// TIA Portal V16 export
// export: Created 2021-11-12T13:32:15.9169285Z, ExportSetting WithDefaults, DisplayName Totally Integrated Automation Portal, DisplayVersion V16 Update 3, DisplayName TIA Portal Version Control Interface, DisplayVersion V16 Update 2, DisplayName TIA Portal Openness, DisplayVersion V16 Update 3, DisplayName SINAMICS Startdrive Advanced, DisplayVersion V16 Update 5, DisplayName SINAMICS Startdrive G130, G150, S120, S150, SINAMICS MV, S210, DisplayVersion V16 Update 5, DisplayName SINAMICS Startdrive G110M, G120, G120C, G120D, G120P, G115D, DisplayVersion V16 Update 5, DisplayName STEP 7 Professional, DisplayVersion V16 Update 3, DisplayName STEP 7 Safety, DisplayVersion V16, DisplayName WinCC UA Professional, DisplayVersion V16 Update 3
FUNCTION_BLOCK "StationBSN2"   // FB15, LAD
{ S7_Optimized_Access := 'TRUE' }
VERSION : 0.1
// stored: AutoNumber true, IsIECCheckEnabled false, IsRetainMemResEnabled false, MemoryReserve 100, SetENOAutomatically false, UDAEnableTagReadback false
   VAR_INPUT
      IS_Inputs : "UDT_COMM_BSN2_CRS";
   END_VAR
   VAR_OUTPUT
      OS_Outputs : "UDT_COMM_CRS_BSN2";
      OS_Status : "UDT_BSN12_Status_specific";
   END_VAR
   VAR
      SF_Alarm1 : "STD_DI_Mon";
      SF_Alarm2 : "STD_DI_Mon";
      SF_Alarm3 : "STD_DI_Mon";
      SF_Alarm4 : "STD_DI_Mon";
      SF_Alarm5 : "STD_DI_Mon";
      SF_Alarm6 : "STD_DI_Mon";
      SF_Alarm7 : "STD_DI_Mon";
      SF_Alarm8 : "STD_DI_Mon";
      SS_Edge : Array[0..15] of Bool;   // Edge evalution
      SS_ParamTemp : Struct
         PartType : Int;   // Production type
         SPTactTime : Int := 0;   // setpoint tact time [s]
         SPStepLength : Int := 0;   // setpoint step length
         SPBurnerHigh : Int := 0;   // setpoint burner high [mm]
         SPTempSetpointZ1 : Int := 0;   // temperature setpoint in zone 1 [°C]
         SPTempSetpointZ2 : Int := 0;   // temperature setpoint in zone 2 [°C]
         SPTempSetpointZ3 : Int := 0;   // temperature setpoint in zone 3 [°C]
         SPTempSetpointZ4 : Int := 0;   // temperature setpoint in zone 4 [°C]
         SPTempSetpointZ5 : Int := 0;   // temperature setpoint in zone 5 [°C]
      END_STRUCT;
      SS_RobotZones : "STD_RobotZones";
      SDIPartID : DInt;
      SI_PartType : Int;
      SI_EjectPartPos { ExternalAccessible := 'False'; ExternalVisible := 'False'; ExternalWritable := 'False'} : Int;   // Position of ejected part
      SB1BlockMapMove : Bool;   // Block transfer datas in map when comm error
      SB1ReqBlockBeltMtion : Bool;   // Button request to block belt motion
      SB1ReqBlockBeltMtion_Aux : Bool;
      SB1ParamChanged : Bool;   // Production paramaters changed trigger
      SB1ReqOnePart { ExternalAccessible := 'False'; ExternalVisible := 'False'; ExternalWritable := 'False'} : Bool;   // Request to eject one part
      SB1ReqAllParts { ExternalAccessible := 'False'; ExternalVisible := 'False'; ExternalWritable := 'False'} : Bool;   // Request to eject all parts in row
      SB1PartEjected : Bool;   // Part ejected memory
      SB1RowEjected : Bool;   // Whole row ejected memory
      SF_TOF_ClearDelay { S7_SetPoint := 'True'} : TOF_TIME;
   END_VAR
   VAR_TEMP
      TS_ParamTemp : Struct
         PartType : Int;   // Production type
         SPTactTime : Int;   // setpoint tact time [s]
         SPStepLength : Int;   // setpoint step length
         SPBurnerHigh : Int;   // setpoint burner high [mm]
         SPTempSetpointZ1 : Int;   // temperature setpoint in zone 1 [°C]
         SPTempSetpointZ2 : Int;   // temperature setpoint in zone 2 [°C]
         SPTempSetpointZ3 : Int;   // temperature setpoint in zone 3 [°C]
         SPTempSetpointZ4 : Int;   // temperature setpoint in zone 4 [°C]
         SPTempSetpointZ5 : Int;   // temperature setpoint in zone 5 [°C]
      END_STRUCT;
      TS_CmdEject : Array[1..5] of Bool;
      TS_EjectSelPreset : Array[1..5] of Byte;
      TS_Part : "UDT_MatCard";
      TDITimeInFurnace_ms : DInt;
      TI_RowNr : Int;   // Transfer mat card according to row number
      TI_BufferFreePos : Int;   // Number of free position in buffer
      TB1PwrOk : Bool;
      TB1BeltMtionBlock : Bool;   // Belt motion blocking
      TB1ReqBlockBeltMtion : Bool;
      TB1SetParam : Bool;   // Set loaded parameters memory
      TB1FreePosBSN : Bool;   // Free position in furnace was found
   END_VAR
   VAR CONSTANT
      CI_FirstRowInsideOven : Int := 8;
      CI_LastRow : Int := 225;
   END_VAR
   // // IS_Inputs.Eject1Up : bsn2 - ejector 1 upper position
   // // IS_Inputs.Eject2Up : bsn2 - ejector 2 upper position
   // // IS_Inputs.Eject3Up : bsn2 - ejector 3 upper position
   // // IS_Inputs.Eject4Up : bsn2 - ejector 4 upper position
   // // IS_Inputs.Eject5Up : bsn2 - ejector 5 upper position
   // // TS_Part.TimeBSN4_s : Time in bsn2 (s)
   VAR_TEMP   // added for the SCL form of the ladder/FBD networks
      _w1 : Bool;
      _w2 : Bool;
      _w3 : Bool;
      _w4 : Bool;
      _w5 : Bool;
      _w6 : Bool;
      _w7 : Bool;
      _w8 : Bool;
      _w9 : Bool;
      _w10 : Bool;
      _w11 : Bool;
      _w12 : Bool;
      _w13 : Bool;
      _w14 : Bool;
      _w15 : Bool;
      _w16 : Bool;
      _w17 : Bool;
      _w18 : Bool;
      _w19 : Bool;
      _w20 : Bool;
      _w21 : Bool;
      _w22 : Bool;
      _w23 : Bool;
      _w24 : Bool;
      _w25 : Bool;
      _w26 : Bool;
   END_VAR
BEGIN

REGION Network 1: *************** Alarms ***************
END_REGION

REGION Network 2: Power OK
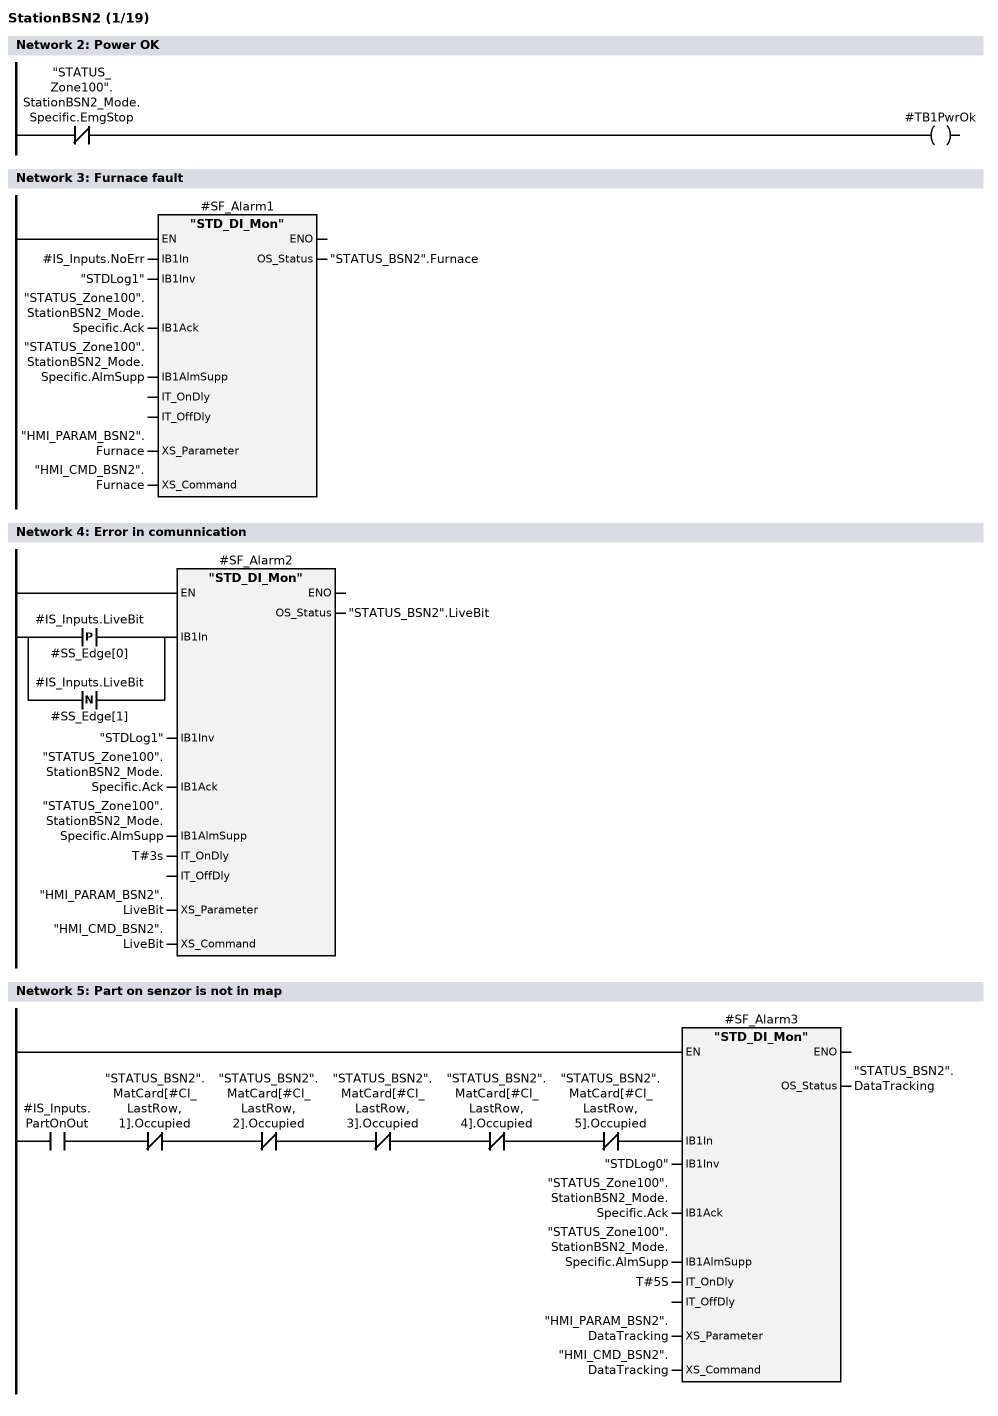
   RUNG wire#powerrail
      I_Contact( "STATUS_Zone100".StationBSN2_Mode.Specific.EmgStop )
      Coil( #TB1PwrOk )
   END_RUNG
   // the same network as SCL:
   #TB1PwrOk := NOT "STATUS_Zone100".StationBSN2_Mode.Specific.EmgStop;
END_REGION

REGION Network 3: Furnace fault
   RUNG wire#powerrail
      #SF_Alarm1(IB1In := #IS_Inputs.NoErr, IB1Inv := "STDLog1", IB1Ack := "STATUS_Zone100".StationBSN2_Mode.Specific.Ack, IB1AlmSupp := "STATUS_Zone100".StationBSN2_Mode.Specific.AlmSupp, IT_OnDly :=, IT_OffDly :=, XS_Parameter := "HMI_PARAM_BSN2".Furnace, XS_Command := "HMI_CMD_BSN2".Furnace, OS_Status => "STATUS_BSN2".Furnace)
   END_RUNG
   // the same network as SCL:
   #SF_Alarm1(IB1In := #IS_Inputs.NoErr,   // "STD_DI_Mon"
              IB1Inv := "STDLog1",
              IB1Ack := "STATUS_Zone100".StationBSN2_Mode.Specific.Ack,
              IB1AlmSupp := "STATUS_Zone100".StationBSN2_Mode.Specific.AlmSupp,
              XS_Parameter := "HMI_PARAM_BSN2".Furnace,
              XS_Command := "HMI_CMD_BSN2".Furnace,
              OS_Status => "STATUS_BSN2".Furnace);
END_REGION

REGION Network 4: Error in comunnication
   RUNG wire#powerrail
      #SF_Alarm2(IB1In := wire#w1, IB1Inv := "STDLog1", IB1Ack := "STATUS_Zone100".StationBSN2_Mode.Specific.Ack, IB1AlmSupp := "STATUS_Zone100".StationBSN2_Mode.Specific.AlmSupp, IT_OnDly := T#3s, IT_OffDly :=, XS_Parameter := "HMI_PARAM_BSN2".LiveBit, XS_Command := "HMI_CMD_BSN2".LiveBit, OS_Status => "STATUS_BSN2".LiveBit)
   END_RUNG
   RUNG wire#powerrail
      P_Contact(operand := #IS_Inputs.LiveBit, bit := #SS_Edge[0])
   END_RUNG wire#w1
   RUNG wire#powerrail
      N_Contact(operand := #IS_Inputs.LiveBit, bit := #SS_Edge[1])
   END_RUNG wire#w1
   // the same network as SCL:
   #_w1 := #IS_Inputs.LiveBit AND NOT #SS_Edge[0];   // rising edge of #IS_Inputs.LiveBit
   #SS_Edge[0] := #IS_Inputs.LiveBit;
   #_w2 := NOT #IS_Inputs.LiveBit AND #SS_Edge[1];   // falling edge of #IS_Inputs.LiveBit
   #SS_Edge[1] := #IS_Inputs.LiveBit;
   #SF_Alarm2(IB1In := #_w1 OR #_w2,   // "STD_DI_Mon"
              IB1Inv := "STDLog1",
              IB1Ack := "STATUS_Zone100".StationBSN2_Mode.Specific.Ack,
              IB1AlmSupp := "STATUS_Zone100".StationBSN2_Mode.Specific.AlmSupp,
              IT_OnDly := T#3s,
              XS_Parameter := "HMI_PARAM_BSN2".LiveBit,
              XS_Command := "HMI_CMD_BSN2".LiveBit,
              OS_Status => "STATUS_BSN2".LiveBit);
END_REGION

REGION Network 5: Part on senzor is not in map
   RUNG wire#powerrail
      #SF_Alarm3(IB1In := wire#w1, IB1Inv := "STDLog0", IB1Ack := "STATUS_Zone100".StationBSN2_Mode.Specific.Ack, IB1AlmSupp := "STATUS_Zone100".StationBSN2_Mode.Specific.AlmSupp, IT_OnDly := T#5S, IT_OffDly :=, XS_Parameter := "HMI_PARAM_BSN2".DataTracking, XS_Command := "HMI_CMD_BSN2".DataTracking, OS_Status => "STATUS_BSN2".DataTracking)
   END_RUNG
   RUNG wire#powerrail
      Contact( #IS_Inputs.PartOnOut )
      I_Contact( "STATUS_BSN2".MatCard[#CI_LastRow, 1].Occupied )
      I_Contact( "STATUS_BSN2".MatCard[#CI_LastRow, 2].Occupied )
      I_Contact( "STATUS_BSN2".MatCard[#CI_LastRow, 3].Occupied )
      I_Contact( "STATUS_BSN2".MatCard[#CI_LastRow, 4].Occupied )
      I_Contact( "STATUS_BSN2".MatCard[#CI_LastRow, 5].Occupied )
   END_RUNG wire#w1
   // the same network as SCL:
   #SF_Alarm3(IB1In := #IS_Inputs.PartOnOut AND NOT "STATUS_BSN2".MatCard[#CI_LastRow, 1].Occupied AND NOT "STATUS_BSN2".MatCard[#CI_LastRow, 2].Occupied AND NOT "STATUS_BSN2".MatCard[#CI_LastRow, 3].Occupied AND NOT "STATUS_BSN2".MatCard[#CI_LastRow, 4].Occupied AND NOT "STATUS_BSN2".MatCard[#CI_LastRow, 5].Occupied,   // "STD_DI_Mon"
              IB1Inv := "STDLog0",
              IB1Ack := "STATUS_Zone100".StationBSN2_Mode.Specific.Ack,
              IB1AlmSupp := "STATUS_Zone100".StationBSN2_Mode.Specific.AlmSupp,
              IT_OnDly := T#5S,
              XS_Parameter := "HMI_PARAM_BSN2".DataTracking,
              XS_Command := "HMI_CMD_BSN2".DataTracking,
              OS_Status => "STATUS_BSN2".DataTracking);
END_REGION

REGION Network 6: Part in map is not on senzor
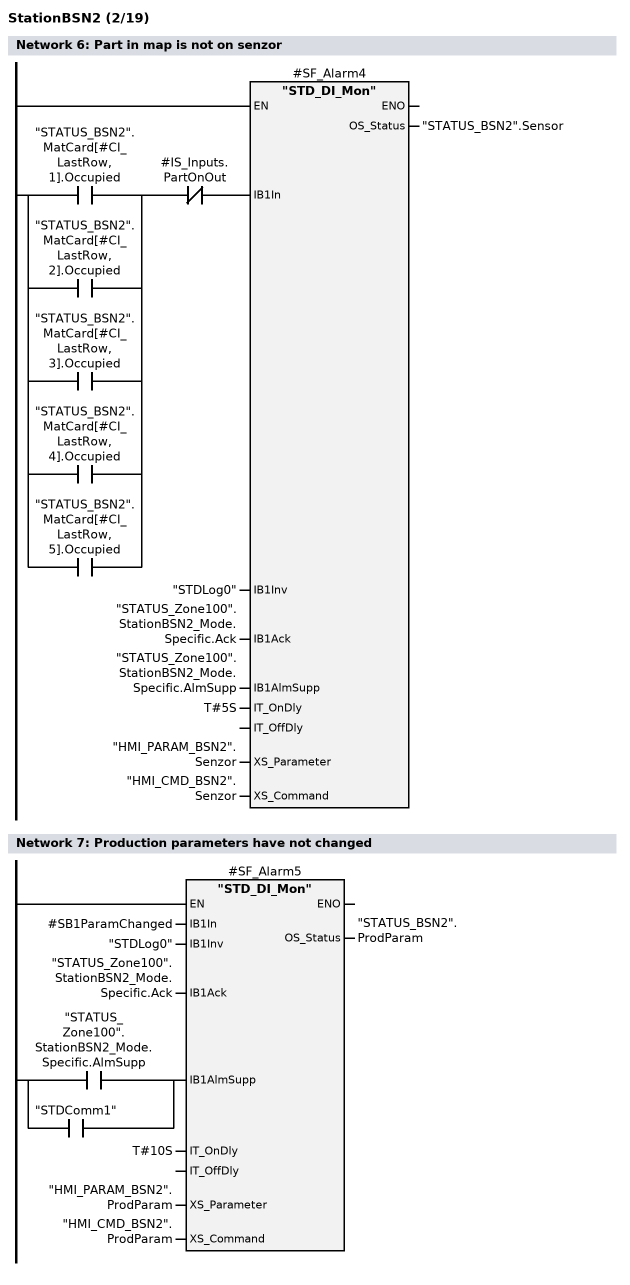
   RUNG wire#powerrail
      #SF_Alarm4(IB1In := wire#w2, IB1Inv := "STDLog0", IB1Ack := "STATUS_Zone100".StationBSN2_Mode.Specific.Ack, IB1AlmSupp := "STATUS_Zone100".StationBSN2_Mode.Specific.AlmSupp, IT_OnDly := T#5S, IT_OffDly :=, XS_Parameter := "HMI_PARAM_BSN2".Senzor, XS_Command := "HMI_CMD_BSN2".Senzor, OS_Status => "STATUS_BSN2".Sensor)
   END_RUNG
   RUNG wire#powerrail
      Contact( "STATUS_BSN2".MatCard[#CI_LastRow, 1].Occupied )
      wire#w1
      I_Contact( #IS_Inputs.PartOnOut )
   END_RUNG wire#w2
   RUNG wire#powerrail
      Contact( "STATUS_BSN2".MatCard[#CI_LastRow, 2].Occupied )
   END_RUNG wire#w1
   RUNG wire#powerrail
      Contact( "STATUS_BSN2".MatCard[#CI_LastRow, 3].Occupied )
   END_RUNG wire#w1
   RUNG wire#powerrail
      Contact( "STATUS_BSN2".MatCard[#CI_LastRow, 4].Occupied )
   END_RUNG wire#w1
   RUNG wire#powerrail
      Contact( "STATUS_BSN2".MatCard[#CI_LastRow, 5].Occupied )
   END_RUNG wire#w1
   // the same network as SCL:
   #SF_Alarm4(IB1In := ("STATUS_BSN2".MatCard[#CI_LastRow, 1].Occupied OR "STATUS_BSN2".MatCard[#CI_LastRow, 2].Occupied OR "STATUS_BSN2".MatCard[#CI_LastRow, 3].Occupied OR "STATUS_BSN2".MatCard[#CI_LastRow, 4].Occupied OR "STATUS_BSN2".MatCard[#CI_LastRow, 5].Occupied) AND NOT #IS_Inputs.PartOnOut,   // "STD_DI_Mon"
              IB1Inv := "STDLog0",
              IB1Ack := "STATUS_Zone100".StationBSN2_Mode.Specific.Ack,
              IB1AlmSupp := "STATUS_Zone100".StationBSN2_Mode.Specific.AlmSupp,
              IT_OnDly := T#5S,
              XS_Parameter := "HMI_PARAM_BSN2".Senzor,
              XS_Command := "HMI_CMD_BSN2".Senzor,
              OS_Status => "STATUS_BSN2".Sensor);
END_REGION

REGION Network 7: Production parameters have not changed
   RUNG wire#powerrail
      #SF_Alarm5(IB1AlmSupp := wire#w1, IB1In := #SB1ParamChanged, IB1Inv := "STDLog0", IB1Ack := "STATUS_Zone100".StationBSN2_Mode.Specific.Ack, IT_OnDly := T#10S, IT_OffDly :=, XS_Parameter := "HMI_PARAM_BSN2".ProdParam, XS_Command := "HMI_CMD_BSN2".ProdParam, OS_Status => "STATUS_BSN2".ProdParam)
   END_RUNG
   RUNG wire#powerrail
      Contact( "STATUS_Zone100".StationBSN2_Mode.Specific.AlmSupp )
   END_RUNG wire#w1
   RUNG wire#powerrail
      Contact( "STDComm1" )
   END_RUNG wire#w1
   // the same network as SCL:
   #SF_Alarm5(IB1In := #SB1ParamChanged,   // "STD_DI_Mon"
              IB1Inv := "STDLog0",
              IB1Ack := "STATUS_Zone100".StationBSN2_Mode.Specific.Ack,
              IB1AlmSupp := "STATUS_Zone100".StationBSN2_Mode.Specific.AlmSupp OR "STDComm1",
              IT_OnDly := T#10S,
              XS_Parameter := "HMI_PARAM_BSN2".ProdParam,
              XS_Command := "HMI_CMD_BSN2".ProdParam,
              OS_Status => "STATUS_BSN2".ProdParam);
END_REGION

REGION Network 8: Long time without step
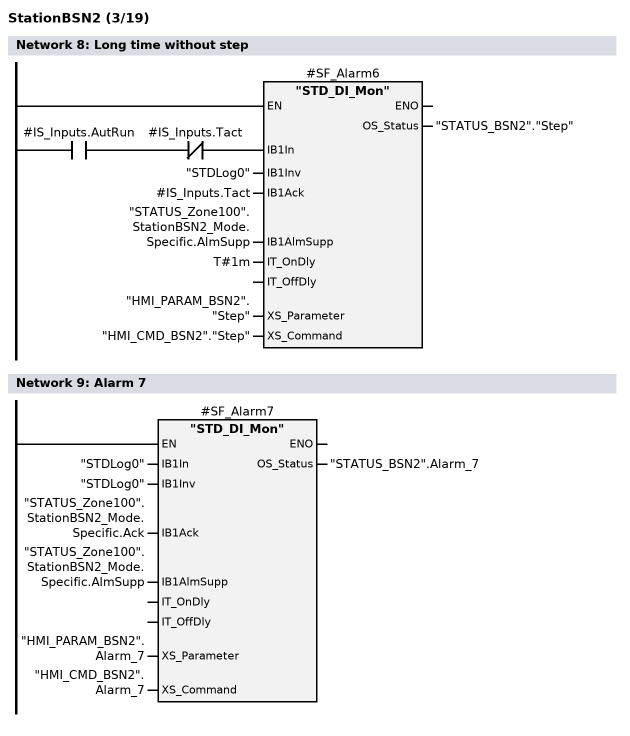
   RUNG wire#powerrail
      #SF_Alarm6(IB1In := wire#w1, IB1Inv := "STDLog0", IB1Ack := #IS_Inputs.Tact, IB1AlmSupp := "STATUS_Zone100".StationBSN2_Mode.Specific.AlmSupp, IT_OnDly := T#1m, IT_OffDly :=, XS_Parameter := "HMI_PARAM_BSN2"."Step", XS_Command := "HMI_CMD_BSN2"."Step", OS_Status => "STATUS_BSN2"."Step")
   END_RUNG
   RUNG wire#powerrail
      Contact( #IS_Inputs.AutRun )
      I_Contact( #IS_Inputs.Tact )
   END_RUNG wire#w1
   // the same network as SCL:
   #SF_Alarm6(IB1In := #IS_Inputs.AutRun AND NOT #IS_Inputs.Tact,   // "STD_DI_Mon"
              IB1Inv := "STDLog0",
              IB1Ack := #IS_Inputs.Tact,
              IB1AlmSupp := "STATUS_Zone100".StationBSN2_Mode.Specific.AlmSupp,
              IT_OnDly := T#1m,
              XS_Parameter := "HMI_PARAM_BSN2"."Step",
              XS_Command := "HMI_CMD_BSN2"."Step",
              OS_Status => "STATUS_BSN2"."Step");
END_REGION

REGION Network 9: Alarm 7
   RUNG wire#powerrail
      #SF_Alarm7(IB1In := "STDLog0", IB1Inv := "STDLog0", IB1Ack := "STATUS_Zone100".StationBSN2_Mode.Specific.Ack, IB1AlmSupp := "STATUS_Zone100".StationBSN2_Mode.Specific.AlmSupp, IT_OnDly :=, IT_OffDly :=, XS_Parameter := "HMI_PARAM_BSN2".Alarm_7, XS_Command := "HMI_CMD_BSN2".Alarm_7, OS_Status => "STATUS_BSN2".Alarm_7)
   END_RUNG
   // the same network as SCL:
   #SF_Alarm7(IB1In := "STDLog0",   // "STD_DI_Mon"
              IB1Inv := "STDLog0",
              IB1Ack := "STATUS_Zone100".StationBSN2_Mode.Specific.Ack,
              IB1AlmSupp := "STATUS_Zone100".StationBSN2_Mode.Specific.AlmSupp,
              XS_Parameter := "HMI_PARAM_BSN2".Alarm_7,
              XS_Command := "HMI_CMD_BSN2".Alarm_7,
              OS_Status => "STATUS_BSN2".Alarm_7);
END_REGION

REGION Network 10: *************** States ***************
END_REGION

REGION Network 11: Temperature, belt extension, ejectors, belt movement
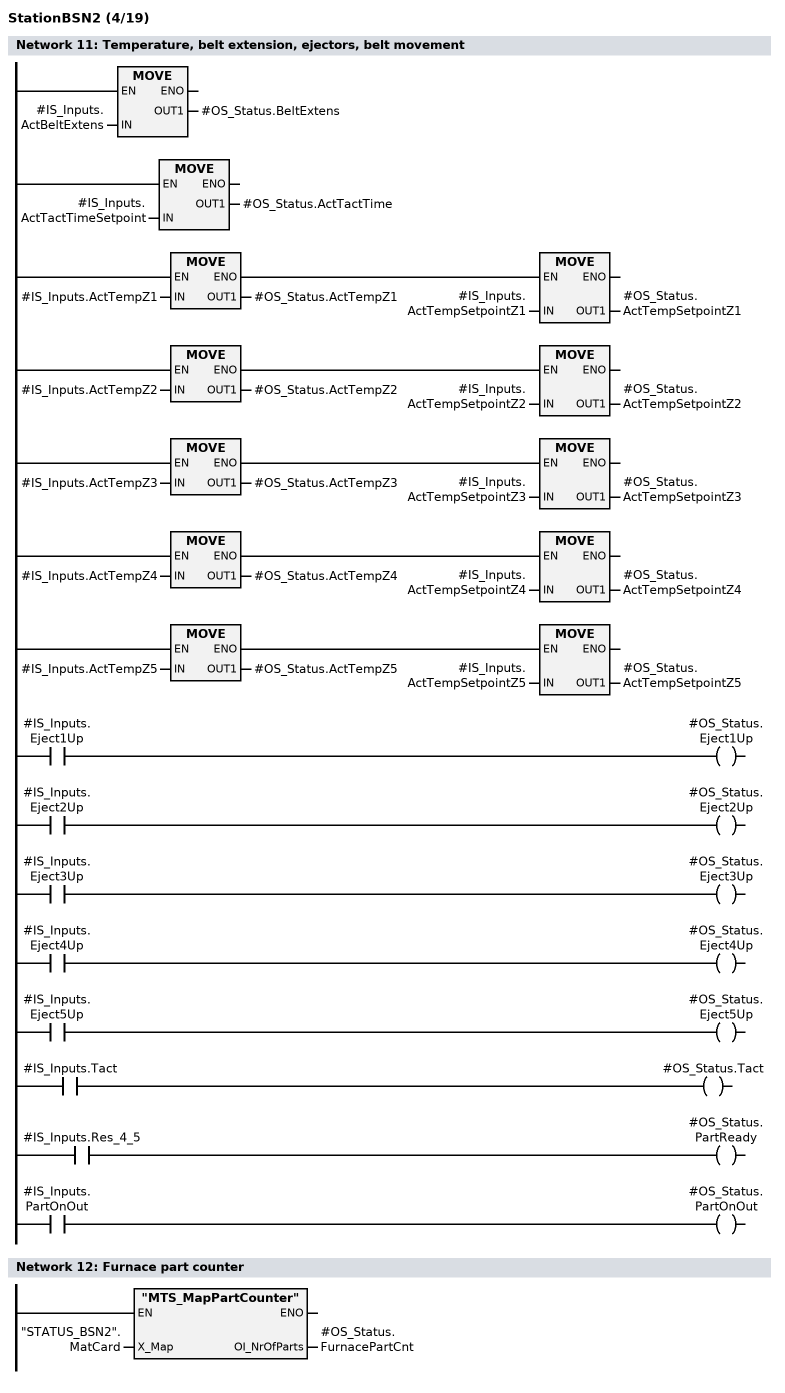
   RUNG wire#powerrail
      Move(in := #IS_Inputs.ActBeltExtens, out1 => #OS_Status.BeltExtens)
   END_RUNG
   RUNG wire#powerrail
      Move(in := #IS_Inputs.ActTactTimeSetpoint, out1 => #OS_Status.ActTactTime)
   END_RUNG
   RUNG wire#powerrail
      Move(in := #IS_Inputs.ActTempZ1, out1 => #OS_Status.ActTempZ1)
      Move(in := #IS_Inputs.ActTempSetpointZ1, out1 => #OS_Status.ActTempSetpointZ1)
   END_RUNG
   RUNG wire#powerrail
      Move(in := #IS_Inputs.ActTempZ2, out1 => #OS_Status.ActTempZ2)
      Move(in := #IS_Inputs.ActTempSetpointZ2, out1 => #OS_Status.ActTempSetpointZ2)
   END_RUNG
   RUNG wire#powerrail
      Move(in := #IS_Inputs.ActTempZ3, out1 => #OS_Status.ActTempZ3)
      Move(in := #IS_Inputs.ActTempSetpointZ3, out1 => #OS_Status.ActTempSetpointZ3)
   END_RUNG
   RUNG wire#powerrail
      Move(in := #IS_Inputs.ActTempZ4, out1 => #OS_Status.ActTempZ4)
      Move(in := #IS_Inputs.ActTempSetpointZ4, out1 => #OS_Status.ActTempSetpointZ4)
   END_RUNG
   RUNG wire#powerrail
      Move(in := #IS_Inputs.ActTempZ5, out1 => #OS_Status.ActTempZ5)
      Move(in := #IS_Inputs.ActTempSetpointZ5, out1 => #OS_Status.ActTempSetpointZ5)
   END_RUNG
   RUNG wire#powerrail
      Contact( #IS_Inputs.Eject1Up )
      Coil( #OS_Status.Eject1Up )
   END_RUNG
   RUNG wire#powerrail
      Contact( #IS_Inputs.Eject2Up )
      Coil( #OS_Status.Eject2Up )
   END_RUNG
   RUNG wire#powerrail
      Contact( #IS_Inputs.Eject3Up )
      Coil( #OS_Status.Eject3Up )
   END_RUNG
   RUNG wire#powerrail
      Contact( #IS_Inputs.Eject4Up )
      Coil( #OS_Status.Eject4Up )
   END_RUNG
   RUNG wire#powerrail
      Contact( #IS_Inputs.Eject5Up )
      Coil( #OS_Status.Eject5Up )
   END_RUNG
   RUNG wire#powerrail
      Contact( #IS_Inputs.Tact )
      Coil( #OS_Status.Tact )
   END_RUNG
   RUNG wire#powerrail
      Contact( #IS_Inputs.Res_4_5 )
      Coil( #OS_Status.PartReady )
   END_RUNG
   RUNG wire#powerrail
      Contact( #IS_Inputs.PartOnOut )
      Coil( #OS_Status.PartOnOut )
   END_RUNG
   // the same network as SCL:
   #OS_Status.BeltExtens := #IS_Inputs.ActBeltExtens;
   #OS_Status.ActTactTime := #IS_Inputs.ActTactTimeSetpoint;
   #OS_Status.ActTempZ1 := #IS_Inputs.ActTempZ1;
   #OS_Status.ActTempSetpointZ1 := #IS_Inputs.ActTempSetpointZ1;
   #OS_Status.ActTempZ2 := #IS_Inputs.ActTempZ2;
   #OS_Status.ActTempSetpointZ2 := #IS_Inputs.ActTempSetpointZ2;
   #OS_Status.ActTempZ3 := #IS_Inputs.ActTempZ3;
   #OS_Status.ActTempSetpointZ3 := #IS_Inputs.ActTempSetpointZ3;
   #OS_Status.ActTempZ4 := #IS_Inputs.ActTempZ4;
   #OS_Status.ActTempSetpointZ4 := #IS_Inputs.ActTempSetpointZ4;
   #OS_Status.ActTempZ5 := #IS_Inputs.ActTempZ5;
   #OS_Status.ActTempSetpointZ5 := #IS_Inputs.ActTempSetpointZ5;
   #OS_Status.Eject1Up := #IS_Inputs.Eject1Up;
   #OS_Status.Eject2Up := #IS_Inputs.Eject2Up;
   #OS_Status.Eject3Up := #IS_Inputs.Eject3Up;
   #OS_Status.Eject4Up := #IS_Inputs.Eject4Up;
   #OS_Status.Eject5Up := #IS_Inputs.Eject5Up;
   #OS_Status.Tact := #IS_Inputs.Tact;
   #OS_Status.PartReady := #IS_Inputs.Res_4_5;
   #OS_Status.PartOnOut := #IS_Inputs.PartOnOut;
END_REGION

REGION Network 12: Furnace part counter
   RUNG wire#powerrail
      "MTS_MapPartCounter"(X_Map := "STATUS_BSN2".MatCard, OI_NrOfParts => #OS_Status.FurnacePartCnt)
   END_RUNG
   // the same network as SCL:
   "MTS_MapPartCounter"(X_Map := "STATUS_BSN2".MatCard, OI_NrOfParts => #OS_Status.FurnacePartCnt);
END_REGION

REGION Network 13: Output conveyor part counter
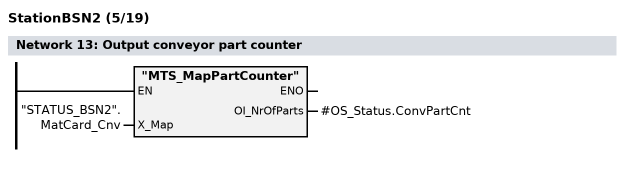
   RUNG wire#powerrail
      "MTS_MapPartCounter"(X_Map := "STATUS_BSN2".MatCard_Cnv, OI_NrOfParts => #OS_Status.ConvPartCnt)
   END_RUNG
   // the same network as SCL:
   "MTS_MapPartCounter"(X_Map := "STATUS_BSN2".MatCard_Cnv, OI_NrOfParts => #OS_Status.ConvPartCnt);
END_REGION

REGION Network 14: *************** Material flow ***************
END_REGION

REGION Network 15: Enable/disable lines
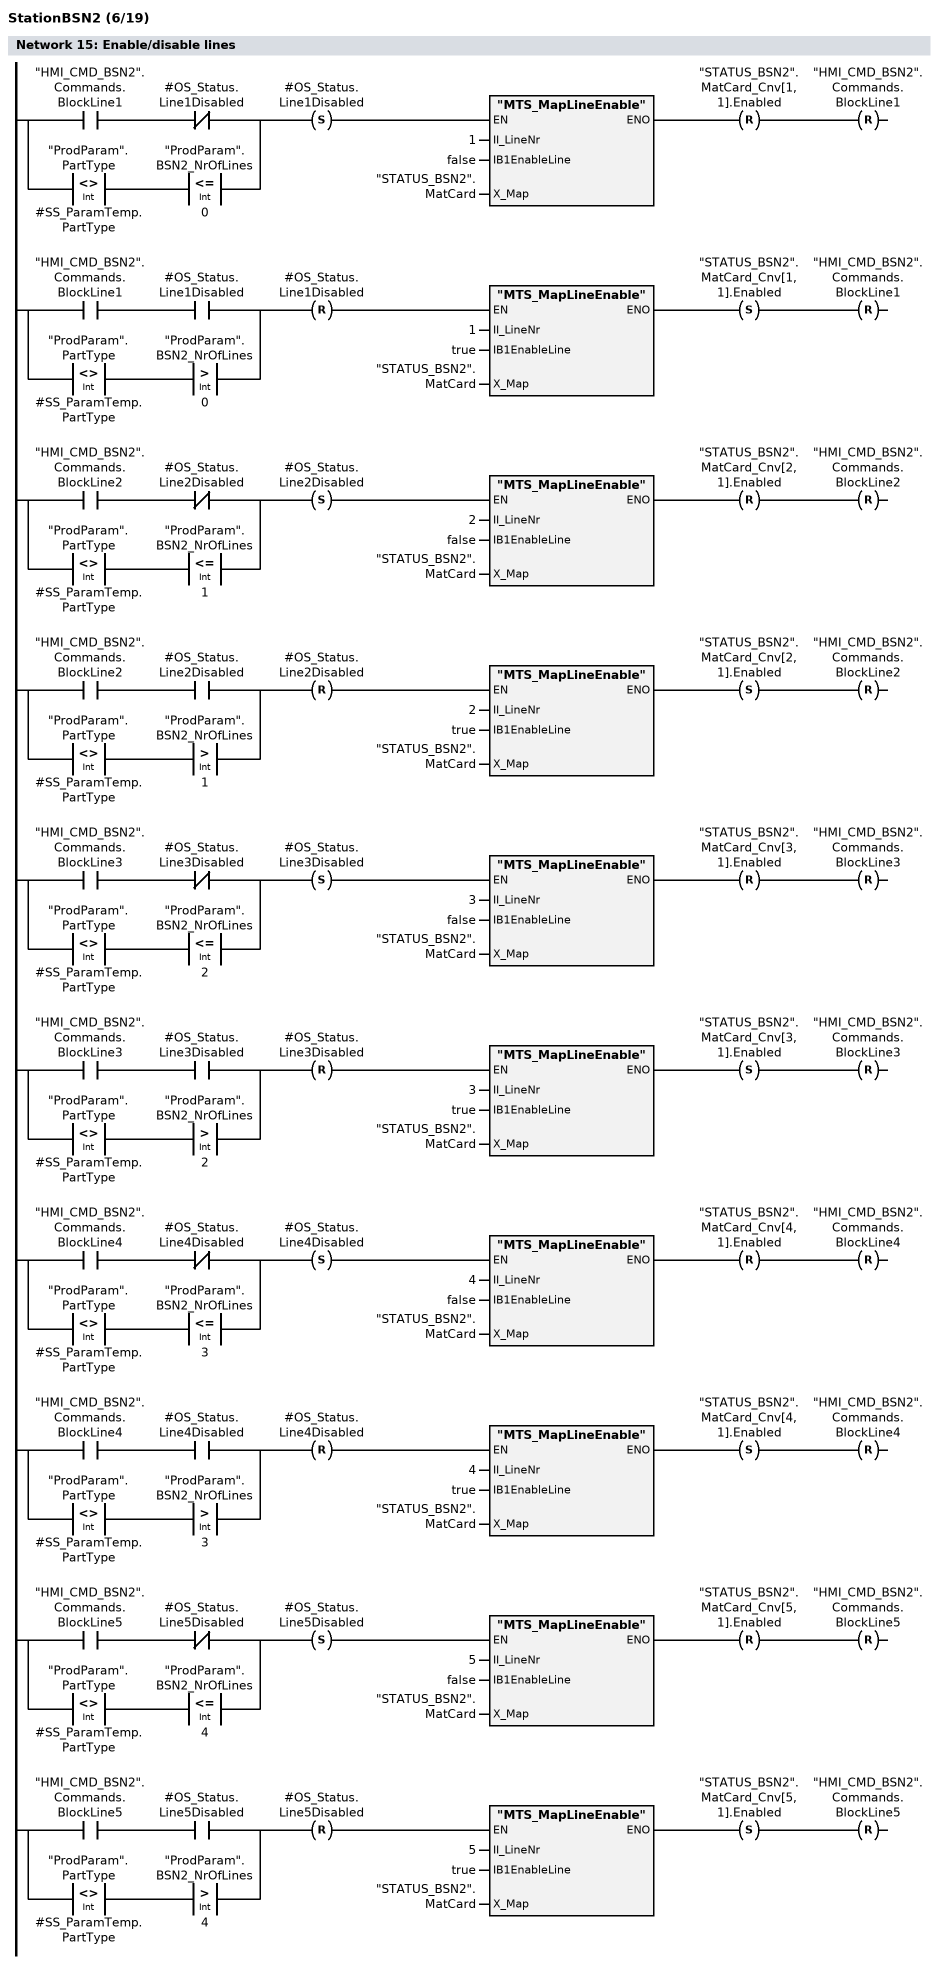
   RUNG wire#powerrail
      Contact( "HMI_CMD_BSN2".Commands.BlockLine1 )
      I_Contact( #OS_Status.Line1Disabled )
      wire#w1
      S_Coil( #OS_Status.Line1Disabled )
      "MTS_MapLineEnable"(II_LineNr := 1, IB1EnableLine := false, X_Map := "STATUS_BSN2".MatCard)
      R_Coil( "STATUS_BSN2".MatCard_Cnv[1, 1].Enabled )
      R_Coil( "HMI_CMD_BSN2".Commands.BlockLine1 )
   END_RUNG
   RUNG wire#powerrail
      { S7_Templates := "SrcType := Int" } NE_Contact(in1 := "ProdParam".PartType, in2 := #SS_ParamTemp.PartType)
      { S7_Templates := "SrcType := Int" } LE_Contact(in1 := "ProdParam".BSN2_NrOfLines, in2 := 0)
   END_RUNG wire#w1
   RUNG wire#powerrail
      Contact( "HMI_CMD_BSN2".Commands.BlockLine1 )
      Contact( #OS_Status.Line1Disabled )
      wire#w2
      R_Coil( #OS_Status.Line1Disabled )
      "MTS_MapLineEnable"(II_LineNr := 1, IB1EnableLine := true, X_Map := "STATUS_BSN2".MatCard)
      S_Coil( "STATUS_BSN2".MatCard_Cnv[1, 1].Enabled )
      R_Coil( "HMI_CMD_BSN2".Commands.BlockLine1 )
   END_RUNG
   RUNG wire#powerrail
      { S7_Templates := "SrcType := Int" } NE_Contact(in1 := "ProdParam".PartType, in2 := #SS_ParamTemp.PartType)
      { S7_Templates := "SrcType := Int" } GT_Contact(in1 := "ProdParam".BSN2_NrOfLines, in2 := 0)
   END_RUNG wire#w2
   RUNG wire#powerrail
      Contact( "HMI_CMD_BSN2".Commands.BlockLine2 )
      I_Contact( #OS_Status.Line2Disabled )
      wire#w3
      S_Coil( #OS_Status.Line2Disabled )
      "MTS_MapLineEnable"(II_LineNr := 2, IB1EnableLine := false, X_Map := "STATUS_BSN2".MatCard)
      R_Coil( "STATUS_BSN2".MatCard_Cnv[2, 1].Enabled )
      R_Coil( "HMI_CMD_BSN2".Commands.BlockLine2 )
   END_RUNG
   RUNG wire#powerrail
      { S7_Templates := "SrcType := Int" } NE_Contact(in1 := "ProdParam".PartType, in2 := #SS_ParamTemp.PartType)
      { S7_Templates := "SrcType := Int" } LE_Contact(in1 := "ProdParam".BSN2_NrOfLines, in2 := 1)
   END_RUNG wire#w3
   RUNG wire#powerrail
      Contact( "HMI_CMD_BSN2".Commands.BlockLine2 )
      Contact( #OS_Status.Line2Disabled )
      wire#w4
      R_Coil( #OS_Status.Line2Disabled )
      "MTS_MapLineEnable"(II_LineNr := 2, IB1EnableLine := true, X_Map := "STATUS_BSN2".MatCard)
      S_Coil( "STATUS_BSN2".MatCard_Cnv[2, 1].Enabled )
      R_Coil( "HMI_CMD_BSN2".Commands.BlockLine2 )
   END_RUNG
   RUNG wire#powerrail
      { S7_Templates := "SrcType := Int" } NE_Contact(in1 := "ProdParam".PartType, in2 := #SS_ParamTemp.PartType)
      { S7_Templates := "SrcType := Int" } GT_Contact(in1 := "ProdParam".BSN2_NrOfLines, in2 := 1)
   END_RUNG wire#w4
   RUNG wire#powerrail
      Contact( "HMI_CMD_BSN2".Commands.BlockLine3 )
      I_Contact( #OS_Status.Line3Disabled )
      wire#w5
      S_Coil( #OS_Status.Line3Disabled )
      "MTS_MapLineEnable"(II_LineNr := 3, IB1EnableLine := false, X_Map := "STATUS_BSN2".MatCard)
      R_Coil( "STATUS_BSN2".MatCard_Cnv[3, 1].Enabled )
      R_Coil( "HMI_CMD_BSN2".Commands.BlockLine3 )
   END_RUNG
   RUNG wire#powerrail
      { S7_Templates := "SrcType := Int" } NE_Contact(in1 := "ProdParam".PartType, in2 := #SS_ParamTemp.PartType)
      { S7_Templates := "SrcType := Int" } LE_Contact(in1 := "ProdParam".BSN2_NrOfLines, in2 := 2)
   END_RUNG wire#w5
   RUNG wire#powerrail
      Contact( "HMI_CMD_BSN2".Commands.BlockLine3 )
      Contact( #OS_Status.Line3Disabled )
      wire#w6
      R_Coil( #OS_Status.Line3Disabled )
      "MTS_MapLineEnable"(II_LineNr := 3, IB1EnableLine := true, X_Map := "STATUS_BSN2".MatCard)
      S_Coil( "STATUS_BSN2".MatCard_Cnv[3, 1].Enabled )
      R_Coil( "HMI_CMD_BSN2".Commands.BlockLine3 )
   END_RUNG
   RUNG wire#powerrail
      { S7_Templates := "SrcType := Int" } NE_Contact(in1 := "ProdParam".PartType, in2 := #SS_ParamTemp.PartType)
      { S7_Templates := "SrcType := Int" } GT_Contact(in1 := "ProdParam".BSN2_NrOfLines, in2 := 2)
   END_RUNG wire#w6
   RUNG wire#powerrail
      Contact( "HMI_CMD_BSN2".Commands.BlockLine4 )
      I_Contact( #OS_Status.Line4Disabled )
      wire#w7
      S_Coil( #OS_Status.Line4Disabled )
      "MTS_MapLineEnable"(II_LineNr := 4, IB1EnableLine := false, X_Map := "STATUS_BSN2".MatCard)
      R_Coil( "STATUS_BSN2".MatCard_Cnv[4, 1].Enabled )
      R_Coil( "HMI_CMD_BSN2".Commands.BlockLine4 )
   END_RUNG
   RUNG wire#powerrail
      { S7_Templates := "SrcType := Int" } NE_Contact(in1 := "ProdParam".PartType, in2 := #SS_ParamTemp.PartType)
      { S7_Templates := "SrcType := Int" } LE_Contact(in1 := "ProdParam".BSN2_NrOfLines, in2 := 3)
   END_RUNG wire#w7
   RUNG wire#powerrail
      Contact( "HMI_CMD_BSN2".Commands.BlockLine4 )
      Contact( #OS_Status.Line4Disabled )
      wire#w8
      R_Coil( #OS_Status.Line4Disabled )
      "MTS_MapLineEnable"(II_LineNr := 4, IB1EnableLine := true, X_Map := "STATUS_BSN2".MatCard)
      S_Coil( "STATUS_BSN2".MatCard_Cnv[4, 1].Enabled )
      R_Coil( "HMI_CMD_BSN2".Commands.BlockLine4 )
   END_RUNG
   RUNG wire#powerrail
      { S7_Templates := "SrcType := Int" } NE_Contact(in1 := "ProdParam".PartType, in2 := #SS_ParamTemp.PartType)
      { S7_Templates := "SrcType := Int" } GT_Contact(in1 := "ProdParam".BSN2_NrOfLines, in2 := 3)
   END_RUNG wire#w8
   RUNG wire#powerrail
      Contact( "HMI_CMD_BSN2".Commands.BlockLine5 )
      I_Contact( #OS_Status.Line5Disabled )
      wire#w9
      S_Coil( #OS_Status.Line5Disabled )
      "MTS_MapLineEnable"(II_LineNr := 5, IB1EnableLine := false, X_Map := "STATUS_BSN2".MatCard)
      R_Coil( "STATUS_BSN2".MatCard_Cnv[5, 1].Enabled )
      R_Coil( "HMI_CMD_BSN2".Commands.BlockLine5 )
   END_RUNG
   RUNG wire#powerrail
      { S7_Templates := "SrcType := Int" } NE_Contact(in1 := "ProdParam".PartType, in2 := #SS_ParamTemp.PartType)
      { S7_Templates := "SrcType := Int" } LE_Contact(in1 := "ProdParam".BSN2_NrOfLines, in2 := 4)
   END_RUNG wire#w9
   RUNG wire#powerrail
      Contact( "HMI_CMD_BSN2".Commands.BlockLine5 )
      Contact( #OS_Status.Line5Disabled )
      wire#w10
      R_Coil( #OS_Status.Line5Disabled )
      "MTS_MapLineEnable"(II_LineNr := 5, IB1EnableLine := true, X_Map := "STATUS_BSN2".MatCard)
      S_Coil( "STATUS_BSN2".MatCard_Cnv[5, 1].Enabled )
      R_Coil( "HMI_CMD_BSN2".Commands.BlockLine5 )
   END_RUNG
   RUNG wire#powerrail
      { S7_Templates := "SrcType := Int" } NE_Contact(in1 := "ProdParam".PartType, in2 := #SS_ParamTemp.PartType)
      { S7_Templates := "SrcType := Int" } GT_Contact(in1 := "ProdParam".BSN2_NrOfLines, in2 := 4)
   END_RUNG wire#w10
   // the same network as SCL:
   #_w1 := ("HMI_CMD_BSN2".Commands.BlockLine1 AND NOT #OS_Status.Line1Disabled) OR (("ProdParam".PartType <> #SS_ParamTemp.PartType) AND ("ProdParam".BSN2_NrOfLines <= 0));
   IF #_w1 THEN #OS_Status.Line1Disabled := TRUE; END_IF;
   "MTS_MapLineEnable"(EN := #_w1,
                       II_LineNr := 1,
                       IB1EnableLine := false,
                       X_Map := "STATUS_BSN2".MatCard,
                       ENO => #_w2);
   IF #_w2 THEN
       "STATUS_BSN2".MatCard_Cnv[1, 1].Enabled := FALSE;
       "HMI_CMD_BSN2".Commands.BlockLine1 := FALSE;
   END_IF;
   #_w3 := ("HMI_CMD_BSN2".Commands.BlockLine1 AND #OS_Status.Line1Disabled) OR (("ProdParam".PartType <> #SS_ParamTemp.PartType) AND ("ProdParam".BSN2_NrOfLines > 0));
   IF #_w3 THEN #OS_Status.Line1Disabled := FALSE; END_IF;
   "MTS_MapLineEnable"(EN := #_w3,
                       II_LineNr := 1,
                       IB1EnableLine := true,
                       X_Map := "STATUS_BSN2".MatCard,
                       ENO => #_w4);
   IF #_w4 THEN
       "STATUS_BSN2".MatCard_Cnv[1, 1].Enabled := TRUE;
       "HMI_CMD_BSN2".Commands.BlockLine1 := FALSE;
   END_IF;
   #_w5 := ("HMI_CMD_BSN2".Commands.BlockLine2 AND NOT #OS_Status.Line2Disabled) OR (("ProdParam".PartType <> #SS_ParamTemp.PartType) AND ("ProdParam".BSN2_NrOfLines <= 1));
   IF #_w5 THEN #OS_Status.Line2Disabled := TRUE; END_IF;
   "MTS_MapLineEnable"(EN := #_w5,
                       II_LineNr := 2,
                       IB1EnableLine := false,
                       X_Map := "STATUS_BSN2".MatCard,
                       ENO => #_w6);
   IF #_w6 THEN
       "STATUS_BSN2".MatCard_Cnv[2, 1].Enabled := FALSE;
       "HMI_CMD_BSN2".Commands.BlockLine2 := FALSE;
   END_IF;
   #_w7 := ("HMI_CMD_BSN2".Commands.BlockLine2 AND #OS_Status.Line2Disabled) OR (("ProdParam".PartType <> #SS_ParamTemp.PartType) AND ("ProdParam".BSN2_NrOfLines > 1));
   IF #_w7 THEN #OS_Status.Line2Disabled := FALSE; END_IF;
   "MTS_MapLineEnable"(EN := #_w7,
                       II_LineNr := 2,
                       IB1EnableLine := true,
                       X_Map := "STATUS_BSN2".MatCard,
                       ENO => #_w8);
   IF #_w8 THEN
       "STATUS_BSN2".MatCard_Cnv[2, 1].Enabled := TRUE;
       "HMI_CMD_BSN2".Commands.BlockLine2 := FALSE;
   END_IF;
   #_w9 := ("HMI_CMD_BSN2".Commands.BlockLine3 AND NOT #OS_Status.Line3Disabled) OR (("ProdParam".PartType <> #SS_ParamTemp.PartType) AND ("ProdParam".BSN2_NrOfLines <= 2));
   IF #_w9 THEN #OS_Status.Line3Disabled := TRUE; END_IF;
   "MTS_MapLineEnable"(EN := #_w9,
                       II_LineNr := 3,
                       IB1EnableLine := false,
                       X_Map := "STATUS_BSN2".MatCard,
                       ENO => #_w10);
   IF #_w10 THEN
       "STATUS_BSN2".MatCard_Cnv[3, 1].Enabled := FALSE;
       "HMI_CMD_BSN2".Commands.BlockLine3 := FALSE;
   END_IF;
   #_w11 := ("HMI_CMD_BSN2".Commands.BlockLine3 AND #OS_Status.Line3Disabled) OR (("ProdParam".PartType <> #SS_ParamTemp.PartType) AND ("ProdParam".BSN2_NrOfLines > 2));
   IF #_w11 THEN #OS_Status.Line3Disabled := FALSE; END_IF;
   "MTS_MapLineEnable"(EN := #_w11,
                       II_LineNr := 3,
                       IB1EnableLine := true,
                       X_Map := "STATUS_BSN2".MatCard,
                       ENO => #_w12);
   IF #_w12 THEN
       "STATUS_BSN2".MatCard_Cnv[3, 1].Enabled := TRUE;
       "HMI_CMD_BSN2".Commands.BlockLine3 := FALSE;
   END_IF;
   #_w13 := ("HMI_CMD_BSN2".Commands.BlockLine4 AND NOT #OS_Status.Line4Disabled) OR (("ProdParam".PartType <> #SS_ParamTemp.PartType) AND ("ProdParam".BSN2_NrOfLines <= 3));
   IF #_w13 THEN #OS_Status.Line4Disabled := TRUE; END_IF;
   "MTS_MapLineEnable"(EN := #_w13,
                       II_LineNr := 4,
                       IB1EnableLine := false,
                       X_Map := "STATUS_BSN2".MatCard,
                       ENO => #_w14);
   IF #_w14 THEN
       "STATUS_BSN2".MatCard_Cnv[4, 1].Enabled := FALSE;
       "HMI_CMD_BSN2".Commands.BlockLine4 := FALSE;
   END_IF;
   #_w15 := ("HMI_CMD_BSN2".Commands.BlockLine4 AND #OS_Status.Line4Disabled) OR (("ProdParam".PartType <> #SS_ParamTemp.PartType) AND ("ProdParam".BSN2_NrOfLines > 3));
   IF #_w15 THEN #OS_Status.Line4Disabled := FALSE; END_IF;
   "MTS_MapLineEnable"(EN := #_w15,
                       II_LineNr := 4,
                       IB1EnableLine := true,
                       X_Map := "STATUS_BSN2".MatCard,
                       ENO => #_w16);
   IF #_w16 THEN
       "STATUS_BSN2".MatCard_Cnv[4, 1].Enabled := TRUE;
       "HMI_CMD_BSN2".Commands.BlockLine4 := FALSE;
   END_IF;
   #_w17 := ("HMI_CMD_BSN2".Commands.BlockLine5 AND NOT #OS_Status.Line5Disabled) OR (("ProdParam".PartType <> #SS_ParamTemp.PartType) AND ("ProdParam".BSN2_NrOfLines <= 4));
   IF #_w17 THEN #OS_Status.Line5Disabled := TRUE; END_IF;
   "MTS_MapLineEnable"(EN := #_w17,
                       II_LineNr := 5,
                       IB1EnableLine := false,
                       X_Map := "STATUS_BSN2".MatCard,
                       ENO => #_w18);
   IF #_w18 THEN
       "STATUS_BSN2".MatCard_Cnv[5, 1].Enabled := FALSE;
       "HMI_CMD_BSN2".Commands.BlockLine5 := FALSE;
   END_IF;
   #_w19 := ("HMI_CMD_BSN2".Commands.BlockLine5 AND #OS_Status.Line5Disabled) OR (("ProdParam".PartType <> #SS_ParamTemp.PartType) AND ("ProdParam".BSN2_NrOfLines > 4));
   IF #_w19 THEN #OS_Status.Line5Disabled := FALSE; END_IF;
   "MTS_MapLineEnable"(EN := #_w19,
                       II_LineNr := 5,
                       IB1EnableLine := true,
                       X_Map := "STATUS_BSN2".MatCard,
                       ENO => #_w20);
   IF #_w20 THEN
       "STATUS_BSN2".MatCard_Cnv[5, 1].Enabled := TRUE;
       "HMI_CMD_BSN2".Commands.BlockLine5 := FALSE;
   END_IF;
END_REGION

REGION Network 16: Set positions in map
   // "JSA0Comm" - change when recipes done
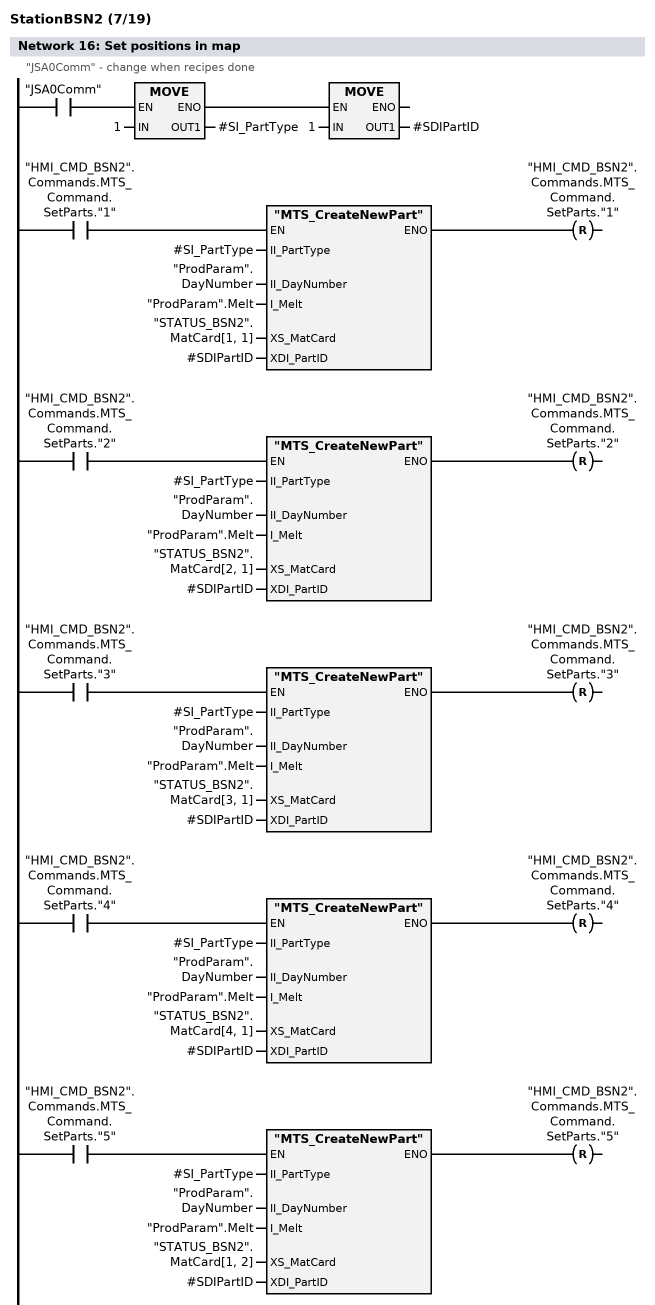
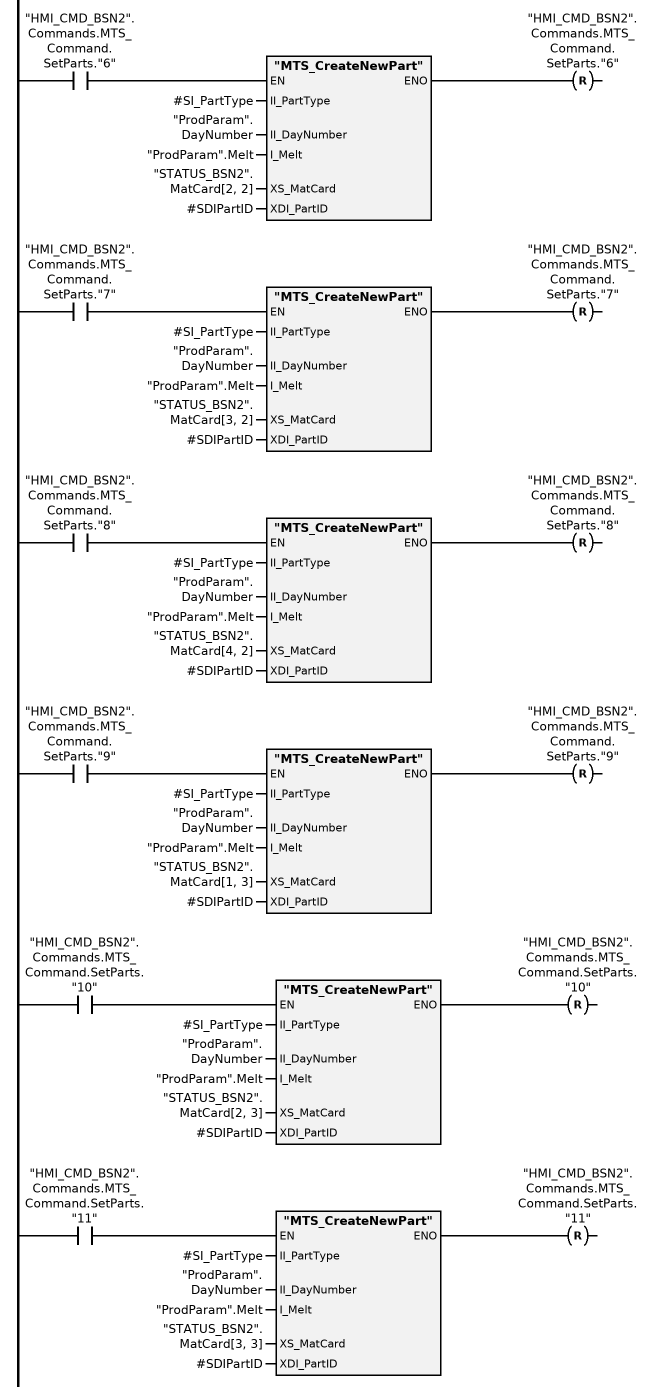
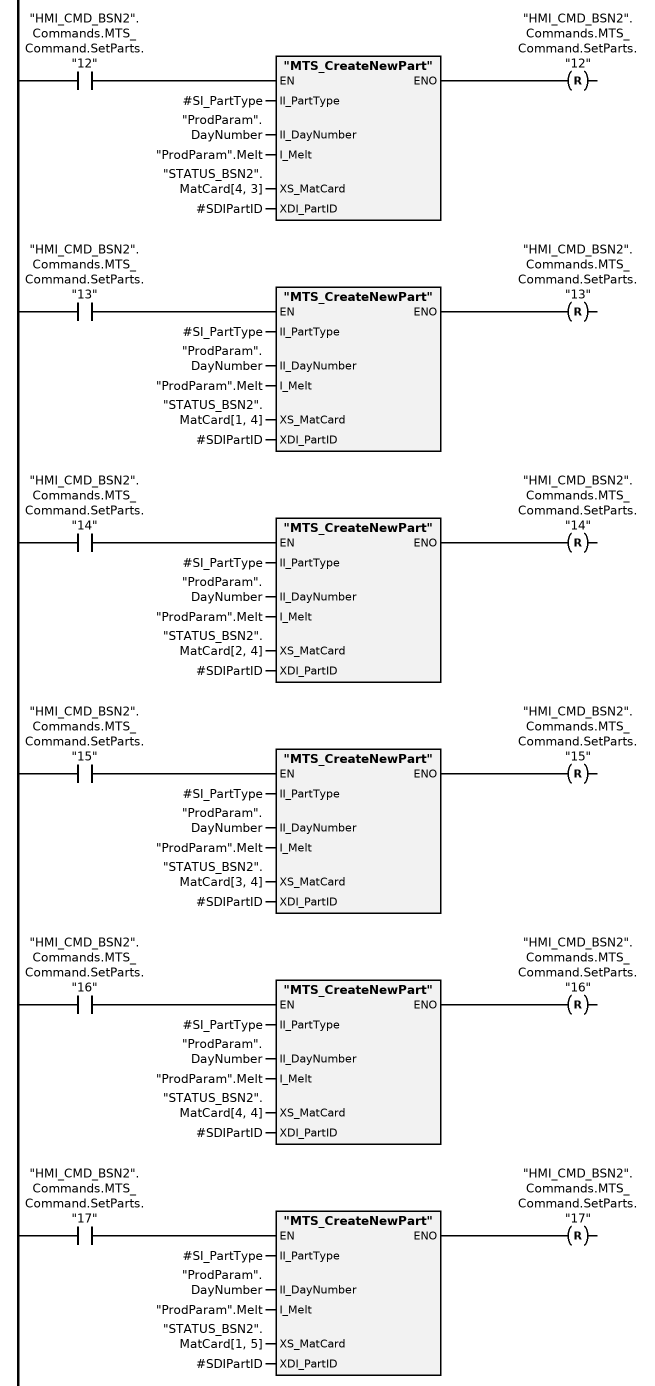
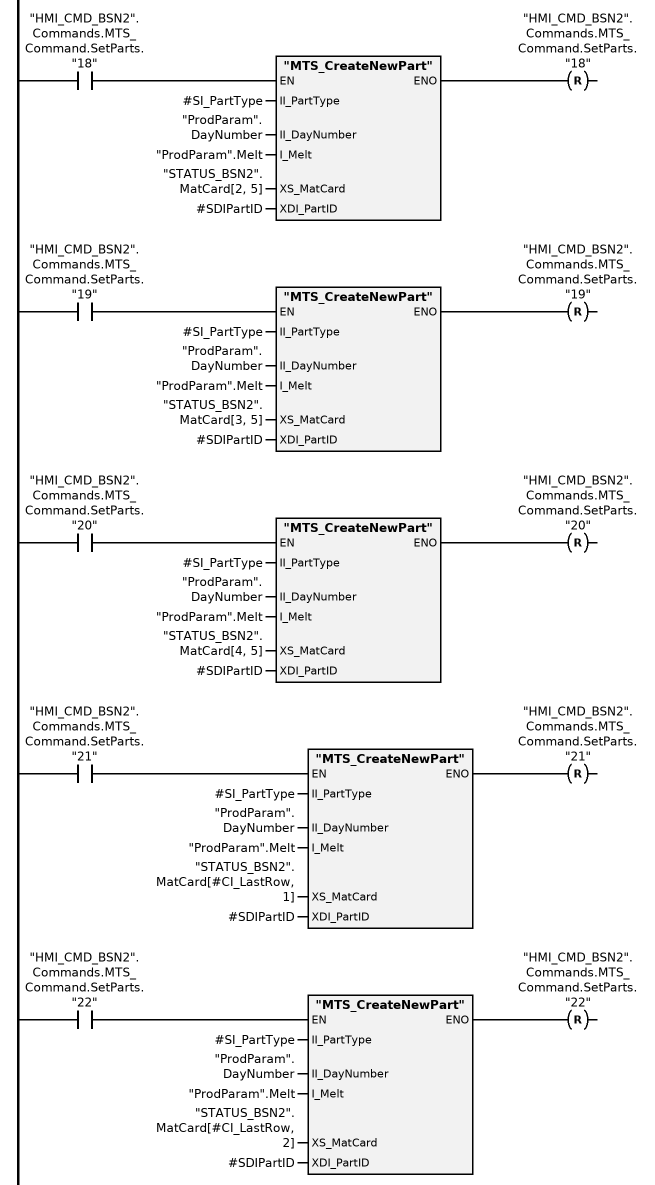
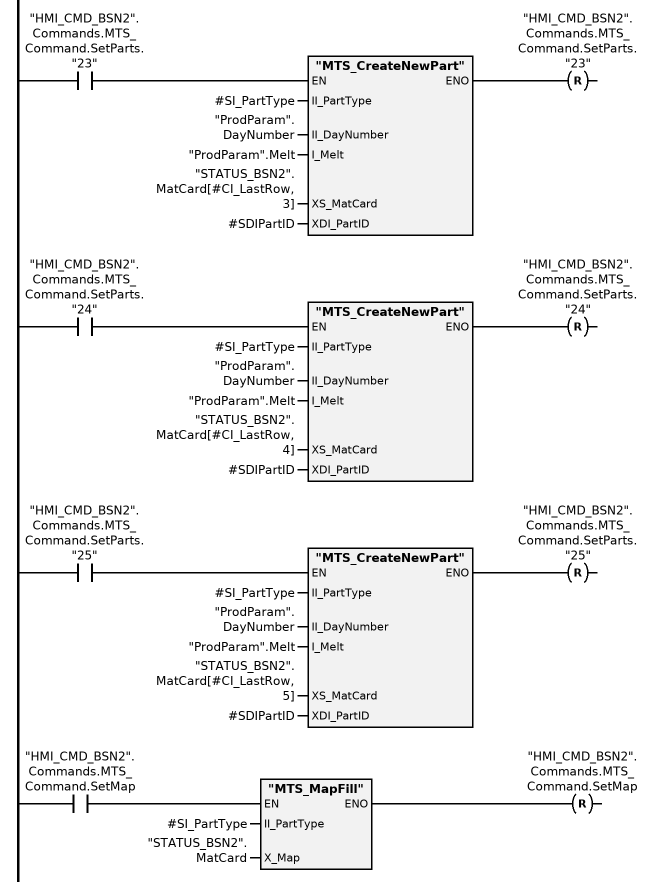
   RUNG wire#powerrail
      Contact( "JSA0Comm" )
      Move(in := 1, out1 => #SI_PartType)
      Move(in := 1, out1 => #SDIPartID)
   END_RUNG
   RUNG wire#powerrail
      Contact( "HMI_CMD_BSN2".Commands.MTS_Command.SetParts."1" )
      "MTS_CreateNewPart"(II_PartType := #SI_PartType, II_DayNumber := "ProdParam".DayNumber, I_Melt := "ProdParam".Melt, XS_MatCard := "STATUS_BSN2".MatCard[1, 1], XDI_PartID := #SDIPartID)
      R_Coil( "HMI_CMD_BSN2".Commands.MTS_Command.SetParts."1" )
   END_RUNG
   RUNG wire#powerrail
      Contact( "HMI_CMD_BSN2".Commands.MTS_Command.SetParts."2" )
      "MTS_CreateNewPart"(II_PartType := #SI_PartType, II_DayNumber := "ProdParam".DayNumber, I_Melt := "ProdParam".Melt, XS_MatCard := "STATUS_BSN2".MatCard[2, 1], XDI_PartID := #SDIPartID)
      R_Coil( "HMI_CMD_BSN2".Commands.MTS_Command.SetParts."2" )
   END_RUNG
   RUNG wire#powerrail
      Contact( "HMI_CMD_BSN2".Commands.MTS_Command.SetParts."3" )
      "MTS_CreateNewPart"(II_PartType := #SI_PartType, II_DayNumber := "ProdParam".DayNumber, I_Melt := "ProdParam".Melt, XS_MatCard := "STATUS_BSN2".MatCard[3, 1], XDI_PartID := #SDIPartID)
      R_Coil( "HMI_CMD_BSN2".Commands.MTS_Command.SetParts."3" )
   END_RUNG
   RUNG wire#powerrail
      Contact( "HMI_CMD_BSN2".Commands.MTS_Command.SetParts."4" )
      "MTS_CreateNewPart"(II_PartType := #SI_PartType, II_DayNumber := "ProdParam".DayNumber, I_Melt := "ProdParam".Melt, XS_MatCard := "STATUS_BSN2".MatCard[4, 1], XDI_PartID := #SDIPartID)
      R_Coil( "HMI_CMD_BSN2".Commands.MTS_Command.SetParts."4" )
   END_RUNG
   RUNG wire#powerrail
      Contact( "HMI_CMD_BSN2".Commands.MTS_Command.SetParts."5" )
      "MTS_CreateNewPart"(II_PartType := #SI_PartType, II_DayNumber := "ProdParam".DayNumber, I_Melt := "ProdParam".Melt, XS_MatCard := "STATUS_BSN2".MatCard[1, 2], XDI_PartID := #SDIPartID)
      R_Coil( "HMI_CMD_BSN2".Commands.MTS_Command.SetParts."5" )
   END_RUNG
   RUNG wire#powerrail
      Contact( "HMI_CMD_BSN2".Commands.MTS_Command.SetParts."6" )
      "MTS_CreateNewPart"(II_PartType := #SI_PartType, II_DayNumber := "ProdParam".DayNumber, I_Melt := "ProdParam".Melt, XS_MatCard := "STATUS_BSN2".MatCard[2, 2], XDI_PartID := #SDIPartID)
      R_Coil( "HMI_CMD_BSN2".Commands.MTS_Command.SetParts."6" )
   END_RUNG
   RUNG wire#powerrail
      Contact( "HMI_CMD_BSN2".Commands.MTS_Command.SetParts."7" )
      "MTS_CreateNewPart"(II_PartType := #SI_PartType, II_DayNumber := "ProdParam".DayNumber, I_Melt := "ProdParam".Melt, XS_MatCard := "STATUS_BSN2".MatCard[3, 2], XDI_PartID := #SDIPartID)
      R_Coil( "HMI_CMD_BSN2".Commands.MTS_Command.SetParts."7" )
   END_RUNG
   RUNG wire#powerrail
      Contact( "HMI_CMD_BSN2".Commands.MTS_Command.SetParts."8" )
      "MTS_CreateNewPart"(II_PartType := #SI_PartType, II_DayNumber := "ProdParam".DayNumber, I_Melt := "ProdParam".Melt, XS_MatCard := "STATUS_BSN2".MatCard[4, 2], XDI_PartID := #SDIPartID)
      R_Coil( "HMI_CMD_BSN2".Commands.MTS_Command.SetParts."8" )
   END_RUNG
   RUNG wire#powerrail
      Contact( "HMI_CMD_BSN2".Commands.MTS_Command.SetParts."9" )
      "MTS_CreateNewPart"(II_PartType := #SI_PartType, II_DayNumber := "ProdParam".DayNumber, I_Melt := "ProdParam".Melt, XS_MatCard := "STATUS_BSN2".MatCard[1, 3], XDI_PartID := #SDIPartID)
      R_Coil( "HMI_CMD_BSN2".Commands.MTS_Command.SetParts."9" )
   END_RUNG
   RUNG wire#powerrail
      Contact( "HMI_CMD_BSN2".Commands.MTS_Command.SetParts."10" )
      "MTS_CreateNewPart"(II_PartType := #SI_PartType, II_DayNumber := "ProdParam".DayNumber, I_Melt := "ProdParam".Melt, XS_MatCard := "STATUS_BSN2".MatCard[2, 3], XDI_PartID := #SDIPartID)
      R_Coil( "HMI_CMD_BSN2".Commands.MTS_Command.SetParts."10" )
   END_RUNG
   RUNG wire#powerrail
      Contact( "HMI_CMD_BSN2".Commands.MTS_Command.SetParts."11" )
      "MTS_CreateNewPart"(II_PartType := #SI_PartType, II_DayNumber := "ProdParam".DayNumber, I_Melt := "ProdParam".Melt, XS_MatCard := "STATUS_BSN2".MatCard[3, 3], XDI_PartID := #SDIPartID)
      R_Coil( "HMI_CMD_BSN2".Commands.MTS_Command.SetParts."11" )
   END_RUNG
   RUNG wire#powerrail
      Contact( "HMI_CMD_BSN2".Commands.MTS_Command.SetParts."12" )
      "MTS_CreateNewPart"(II_PartType := #SI_PartType, II_DayNumber := "ProdParam".DayNumber, I_Melt := "ProdParam".Melt, XS_MatCard := "STATUS_BSN2".MatCard[4, 3], XDI_PartID := #SDIPartID)
      R_Coil( "HMI_CMD_BSN2".Commands.MTS_Command.SetParts."12" )
   END_RUNG
   RUNG wire#powerrail
      Contact( "HMI_CMD_BSN2".Commands.MTS_Command.SetParts."13" )
      "MTS_CreateNewPart"(II_PartType := #SI_PartType, II_DayNumber := "ProdParam".DayNumber, I_Melt := "ProdParam".Melt, XS_MatCard := "STATUS_BSN2".MatCard[1, 4], XDI_PartID := #SDIPartID)
      R_Coil( "HMI_CMD_BSN2".Commands.MTS_Command.SetParts."13" )
   END_RUNG
   RUNG wire#powerrail
      Contact( "HMI_CMD_BSN2".Commands.MTS_Command.SetParts."14" )
      "MTS_CreateNewPart"(II_PartType := #SI_PartType, II_DayNumber := "ProdParam".DayNumber, I_Melt := "ProdParam".Melt, XS_MatCard := "STATUS_BSN2".MatCard[2, 4], XDI_PartID := #SDIPartID)
      R_Coil( "HMI_CMD_BSN2".Commands.MTS_Command.SetParts."14" )
   END_RUNG
   RUNG wire#powerrail
      Contact( "HMI_CMD_BSN2".Commands.MTS_Command.SetParts."15" )
      "MTS_CreateNewPart"(II_PartType := #SI_PartType, II_DayNumber := "ProdParam".DayNumber, I_Melt := "ProdParam".Melt, XS_MatCard := "STATUS_BSN2".MatCard[3, 4], XDI_PartID := #SDIPartID)
      R_Coil( "HMI_CMD_BSN2".Commands.MTS_Command.SetParts."15" )
   END_RUNG
   RUNG wire#powerrail
      Contact( "HMI_CMD_BSN2".Commands.MTS_Command.SetParts."16" )
      "MTS_CreateNewPart"(II_PartType := #SI_PartType, II_DayNumber := "ProdParam".DayNumber, I_Melt := "ProdParam".Melt, XS_MatCard := "STATUS_BSN2".MatCard[4, 4], XDI_PartID := #SDIPartID)
      R_Coil( "HMI_CMD_BSN2".Commands.MTS_Command.SetParts."16" )
   END_RUNG
   RUNG wire#powerrail
      Contact( "HMI_CMD_BSN2".Commands.MTS_Command.SetParts."17" )
      "MTS_CreateNewPart"(II_PartType := #SI_PartType, II_DayNumber := "ProdParam".DayNumber, I_Melt := "ProdParam".Melt, XS_MatCard := "STATUS_BSN2".MatCard[1, 5], XDI_PartID := #SDIPartID)
      R_Coil( "HMI_CMD_BSN2".Commands.MTS_Command.SetParts."17" )
   END_RUNG
   RUNG wire#powerrail
      Contact( "HMI_CMD_BSN2".Commands.MTS_Command.SetParts."18" )
      "MTS_CreateNewPart"(II_PartType := #SI_PartType, II_DayNumber := "ProdParam".DayNumber, I_Melt := "ProdParam".Melt, XS_MatCard := "STATUS_BSN2".MatCard[2, 5], XDI_PartID := #SDIPartID)
      R_Coil( "HMI_CMD_BSN2".Commands.MTS_Command.SetParts."18" )
   END_RUNG
   RUNG wire#powerrail
      Contact( "HMI_CMD_BSN2".Commands.MTS_Command.SetParts."19" )
      "MTS_CreateNewPart"(II_PartType := #SI_PartType, II_DayNumber := "ProdParam".DayNumber, I_Melt := "ProdParam".Melt, XS_MatCard := "STATUS_BSN2".MatCard[3, 5], XDI_PartID := #SDIPartID)
      R_Coil( "HMI_CMD_BSN2".Commands.MTS_Command.SetParts."19" )
   END_RUNG
   RUNG wire#powerrail
      Contact( "HMI_CMD_BSN2".Commands.MTS_Command.SetParts."20" )
      "MTS_CreateNewPart"(II_PartType := #SI_PartType, II_DayNumber := "ProdParam".DayNumber, I_Melt := "ProdParam".Melt, XS_MatCard := "STATUS_BSN2".MatCard[4, 5], XDI_PartID := #SDIPartID)
      R_Coil( "HMI_CMD_BSN2".Commands.MTS_Command.SetParts."20" )
   END_RUNG
   RUNG wire#powerrail
      Contact( "HMI_CMD_BSN2".Commands.MTS_Command.SetParts."21" )
      "MTS_CreateNewPart"(II_PartType := #SI_PartType, II_DayNumber := "ProdParam".DayNumber, I_Melt := "ProdParam".Melt, XS_MatCard := "STATUS_BSN2".MatCard[#CI_LastRow, 1], XDI_PartID := #SDIPartID)
      R_Coil( "HMI_CMD_BSN2".Commands.MTS_Command.SetParts."21" )
   END_RUNG
   RUNG wire#powerrail
      Contact( "HMI_CMD_BSN2".Commands.MTS_Command.SetParts."22" )
      "MTS_CreateNewPart"(II_PartType := #SI_PartType, II_DayNumber := "ProdParam".DayNumber, I_Melt := "ProdParam".Melt, XS_MatCard := "STATUS_BSN2".MatCard[#CI_LastRow, 2], XDI_PartID := #SDIPartID)
      R_Coil( "HMI_CMD_BSN2".Commands.MTS_Command.SetParts."22" )
   END_RUNG
   RUNG wire#powerrail
      Contact( "HMI_CMD_BSN2".Commands.MTS_Command.SetParts."23" )
      "MTS_CreateNewPart"(II_PartType := #SI_PartType, II_DayNumber := "ProdParam".DayNumber, I_Melt := "ProdParam".Melt, XS_MatCard := "STATUS_BSN2".MatCard[#CI_LastRow, 3], XDI_PartID := #SDIPartID)
      R_Coil( "HMI_CMD_BSN2".Commands.MTS_Command.SetParts."23" )
   END_RUNG
   RUNG wire#powerrail
      Contact( "HMI_CMD_BSN2".Commands.MTS_Command.SetParts."24" )
      "MTS_CreateNewPart"(II_PartType := #SI_PartType, II_DayNumber := "ProdParam".DayNumber, I_Melt := "ProdParam".Melt, XS_MatCard := "STATUS_BSN2".MatCard[#CI_LastRow, 4], XDI_PartID := #SDIPartID)
      R_Coil( "HMI_CMD_BSN2".Commands.MTS_Command.SetParts."24" )
   END_RUNG
   RUNG wire#powerrail
      Contact( "HMI_CMD_BSN2".Commands.MTS_Command.SetParts."25" )
      "MTS_CreateNewPart"(II_PartType := #SI_PartType, II_DayNumber := "ProdParam".DayNumber, I_Melt := "ProdParam".Melt, XS_MatCard := "STATUS_BSN2".MatCard[#CI_LastRow, 5], XDI_PartID := #SDIPartID)
      R_Coil( "HMI_CMD_BSN2".Commands.MTS_Command.SetParts."25" )
   END_RUNG
   RUNG wire#powerrail
      Contact( "HMI_CMD_BSN2".Commands.MTS_Command.SetMap )
      "MTS_MapFill"(II_PartType := #SI_PartType, X_Map := "STATUS_BSN2".MatCard)
      R_Coil( "HMI_CMD_BSN2".Commands.MTS_Command.SetMap )
   END_RUNG
   // the same network as SCL:
   IF "JSA0Comm" THEN
       #SI_PartType := 1;
       #SDIPartID := 1;
   END_IF;
   "MTS_CreateNewPart"(EN := "HMI_CMD_BSN2".Commands.MTS_Command.SetParts."1",
                       II_PartType := #SI_PartType,
                       II_DayNumber := "ProdParam".DayNumber,
                       I_Melt := "ProdParam".Melt,
                       XS_MatCard := "STATUS_BSN2".MatCard[1, 1],
                       XDI_PartID := #SDIPartID,
                       ENO => #_w1);
   IF #_w1 THEN "HMI_CMD_BSN2".Commands.MTS_Command.SetParts."1" := FALSE; END_IF;
   "MTS_CreateNewPart"(EN := "HMI_CMD_BSN2".Commands.MTS_Command.SetParts."2",
                       II_PartType := #SI_PartType,
                       II_DayNumber := "ProdParam".DayNumber,
                       I_Melt := "ProdParam".Melt,
                       XS_MatCard := "STATUS_BSN2".MatCard[2, 1],
                       XDI_PartID := #SDIPartID,
                       ENO => #_w2);
   IF #_w2 THEN "HMI_CMD_BSN2".Commands.MTS_Command.SetParts."2" := FALSE; END_IF;
   "MTS_CreateNewPart"(EN := "HMI_CMD_BSN2".Commands.MTS_Command.SetParts."3",
                       II_PartType := #SI_PartType,
                       II_DayNumber := "ProdParam".DayNumber,
                       I_Melt := "ProdParam".Melt,
                       XS_MatCard := "STATUS_BSN2".MatCard[3, 1],
                       XDI_PartID := #SDIPartID,
                       ENO => #_w3);
   IF #_w3 THEN "HMI_CMD_BSN2".Commands.MTS_Command.SetParts."3" := FALSE; END_IF;
   "MTS_CreateNewPart"(EN := "HMI_CMD_BSN2".Commands.MTS_Command.SetParts."4",
                       II_PartType := #SI_PartType,
                       II_DayNumber := "ProdParam".DayNumber,
                       I_Melt := "ProdParam".Melt,
                       XS_MatCard := "STATUS_BSN2".MatCard[4, 1],
                       XDI_PartID := #SDIPartID,
                       ENO => #_w4);
   IF #_w4 THEN "HMI_CMD_BSN2".Commands.MTS_Command.SetParts."4" := FALSE; END_IF;
   "MTS_CreateNewPart"(EN := "HMI_CMD_BSN2".Commands.MTS_Command.SetParts."5",
                       II_PartType := #SI_PartType,
                       II_DayNumber := "ProdParam".DayNumber,
                       I_Melt := "ProdParam".Melt,
                       XS_MatCard := "STATUS_BSN2".MatCard[1, 2],
                       XDI_PartID := #SDIPartID,
                       ENO => #_w5);
   IF #_w5 THEN "HMI_CMD_BSN2".Commands.MTS_Command.SetParts."5" := FALSE; END_IF;
   "MTS_CreateNewPart"(EN := "HMI_CMD_BSN2".Commands.MTS_Command.SetParts."6",
                       II_PartType := #SI_PartType,
                       II_DayNumber := "ProdParam".DayNumber,
                       I_Melt := "ProdParam".Melt,
                       XS_MatCard := "STATUS_BSN2".MatCard[2, 2],
                       XDI_PartID := #SDIPartID,
                       ENO => #_w6);
   IF #_w6 THEN "HMI_CMD_BSN2".Commands.MTS_Command.SetParts."6" := FALSE; END_IF;
   "MTS_CreateNewPart"(EN := "HMI_CMD_BSN2".Commands.MTS_Command.SetParts."7",
                       II_PartType := #SI_PartType,
                       II_DayNumber := "ProdParam".DayNumber,
                       I_Melt := "ProdParam".Melt,
                       XS_MatCard := "STATUS_BSN2".MatCard[3, 2],
                       XDI_PartID := #SDIPartID,
                       ENO => #_w7);
   IF #_w7 THEN "HMI_CMD_BSN2".Commands.MTS_Command.SetParts."7" := FALSE; END_IF;
   "MTS_CreateNewPart"(EN := "HMI_CMD_BSN2".Commands.MTS_Command.SetParts."8",
                       II_PartType := #SI_PartType,
                       II_DayNumber := "ProdParam".DayNumber,
                       I_Melt := "ProdParam".Melt,
                       XS_MatCard := "STATUS_BSN2".MatCard[4, 2],
                       XDI_PartID := #SDIPartID,
                       ENO => #_w8);
   IF #_w8 THEN "HMI_CMD_BSN2".Commands.MTS_Command.SetParts."8" := FALSE; END_IF;
   "MTS_CreateNewPart"(EN := "HMI_CMD_BSN2".Commands.MTS_Command.SetParts."9",
                       II_PartType := #SI_PartType,
                       II_DayNumber := "ProdParam".DayNumber,
                       I_Melt := "ProdParam".Melt,
                       XS_MatCard := "STATUS_BSN2".MatCard[1, 3],
                       XDI_PartID := #SDIPartID,
                       ENO => #_w9);
   IF #_w9 THEN "HMI_CMD_BSN2".Commands.MTS_Command.SetParts."9" := FALSE; END_IF;
   "MTS_CreateNewPart"(EN := "HMI_CMD_BSN2".Commands.MTS_Command.SetParts."10",
                       II_PartType := #SI_PartType,
                       II_DayNumber := "ProdParam".DayNumber,
                       I_Melt := "ProdParam".Melt,
                       XS_MatCard := "STATUS_BSN2".MatCard[2, 3],
                       XDI_PartID := #SDIPartID,
                       ENO => #_w10);
   IF #_w10 THEN "HMI_CMD_BSN2".Commands.MTS_Command.SetParts."10" := FALSE; END_IF;
   "MTS_CreateNewPart"(EN := "HMI_CMD_BSN2".Commands.MTS_Command.SetParts."11",
                       II_PartType := #SI_PartType,
                       II_DayNumber := "ProdParam".DayNumber,
                       I_Melt := "ProdParam".Melt,
                       XS_MatCard := "STATUS_BSN2".MatCard[3, 3],
                       XDI_PartID := #SDIPartID,
                       ENO => #_w11);
   IF #_w11 THEN "HMI_CMD_BSN2".Commands.MTS_Command.SetParts."11" := FALSE; END_IF;
   "MTS_CreateNewPart"(EN := "HMI_CMD_BSN2".Commands.MTS_Command.SetParts."12",
                       II_PartType := #SI_PartType,
                       II_DayNumber := "ProdParam".DayNumber,
                       I_Melt := "ProdParam".Melt,
                       XS_MatCard := "STATUS_BSN2".MatCard[4, 3],
                       XDI_PartID := #SDIPartID,
                       ENO => #_w12);
   IF #_w12 THEN "HMI_CMD_BSN2".Commands.MTS_Command.SetParts."12" := FALSE; END_IF;
   "MTS_CreateNewPart"(EN := "HMI_CMD_BSN2".Commands.MTS_Command.SetParts."13",
                       II_PartType := #SI_PartType,
                       II_DayNumber := "ProdParam".DayNumber,
                       I_Melt := "ProdParam".Melt,
                       XS_MatCard := "STATUS_BSN2".MatCard[1, 4],
                       XDI_PartID := #SDIPartID,
                       ENO => #_w13);
   IF #_w13 THEN "HMI_CMD_BSN2".Commands.MTS_Command.SetParts."13" := FALSE; END_IF;
   "MTS_CreateNewPart"(EN := "HMI_CMD_BSN2".Commands.MTS_Command.SetParts."14",
                       II_PartType := #SI_PartType,
                       II_DayNumber := "ProdParam".DayNumber,
                       I_Melt := "ProdParam".Melt,
                       XS_MatCard := "STATUS_BSN2".MatCard[2, 4],
                       XDI_PartID := #SDIPartID,
                       ENO => #_w14);
   IF #_w14 THEN "HMI_CMD_BSN2".Commands.MTS_Command.SetParts."14" := FALSE; END_IF;
   "MTS_CreateNewPart"(EN := "HMI_CMD_BSN2".Commands.MTS_Command.SetParts."15",
                       II_PartType := #SI_PartType,
                       II_DayNumber := "ProdParam".DayNumber,
                       I_Melt := "ProdParam".Melt,
                       XS_MatCard := "STATUS_BSN2".MatCard[3, 4],
                       XDI_PartID := #SDIPartID,
                       ENO => #_w15);
   IF #_w15 THEN "HMI_CMD_BSN2".Commands.MTS_Command.SetParts."15" := FALSE; END_IF;
   "MTS_CreateNewPart"(EN := "HMI_CMD_BSN2".Commands.MTS_Command.SetParts."16",
                       II_PartType := #SI_PartType,
                       II_DayNumber := "ProdParam".DayNumber,
                       I_Melt := "ProdParam".Melt,
                       XS_MatCard := "STATUS_BSN2".MatCard[4, 4],
                       XDI_PartID := #SDIPartID,
                       ENO => #_w16);
   IF #_w16 THEN "HMI_CMD_BSN2".Commands.MTS_Command.SetParts."16" := FALSE; END_IF;
   "MTS_CreateNewPart"(EN := "HMI_CMD_BSN2".Commands.MTS_Command.SetParts."17",
                       II_PartType := #SI_PartType,
                       II_DayNumber := "ProdParam".DayNumber,
                       I_Melt := "ProdParam".Melt,
                       XS_MatCard := "STATUS_BSN2".MatCard[1, 5],
                       XDI_PartID := #SDIPartID,
                       ENO => #_w17);
   IF #_w17 THEN "HMI_CMD_BSN2".Commands.MTS_Command.SetParts."17" := FALSE; END_IF;
   "MTS_CreateNewPart"(EN := "HMI_CMD_BSN2".Commands.MTS_Command.SetParts."18",
                       II_PartType := #SI_PartType,
                       II_DayNumber := "ProdParam".DayNumber,
                       I_Melt := "ProdParam".Melt,
                       XS_MatCard := "STATUS_BSN2".MatCard[2, 5],
                       XDI_PartID := #SDIPartID,
                       ENO => #_w18);
   IF #_w18 THEN "HMI_CMD_BSN2".Commands.MTS_Command.SetParts."18" := FALSE; END_IF;
   "MTS_CreateNewPart"(EN := "HMI_CMD_BSN2".Commands.MTS_Command.SetParts."19",
                       II_PartType := #SI_PartType,
                       II_DayNumber := "ProdParam".DayNumber,
                       I_Melt := "ProdParam".Melt,
                       XS_MatCard := "STATUS_BSN2".MatCard[3, 5],
                       XDI_PartID := #SDIPartID,
                       ENO => #_w19);
   IF #_w19 THEN "HMI_CMD_BSN2".Commands.MTS_Command.SetParts."19" := FALSE; END_IF;
   "MTS_CreateNewPart"(EN := "HMI_CMD_BSN2".Commands.MTS_Command.SetParts."20",
                       II_PartType := #SI_PartType,
                       II_DayNumber := "ProdParam".DayNumber,
                       I_Melt := "ProdParam".Melt,
                       XS_MatCard := "STATUS_BSN2".MatCard[4, 5],
                       XDI_PartID := #SDIPartID,
                       ENO => #_w20);
   IF #_w20 THEN "HMI_CMD_BSN2".Commands.MTS_Command.SetParts."20" := FALSE; END_IF;
   "MTS_CreateNewPart"(EN := "HMI_CMD_BSN2".Commands.MTS_Command.SetParts."21",
                       II_PartType := #SI_PartType,
                       II_DayNumber := "ProdParam".DayNumber,
                       I_Melt := "ProdParam".Melt,
                       XS_MatCard := "STATUS_BSN2".MatCard[#CI_LastRow, 1],
                       XDI_PartID := #SDIPartID,
                       ENO => #_w21);
   IF #_w21 THEN "HMI_CMD_BSN2".Commands.MTS_Command.SetParts."21" := FALSE; END_IF;
   "MTS_CreateNewPart"(EN := "HMI_CMD_BSN2".Commands.MTS_Command.SetParts."22",
                       II_PartType := #SI_PartType,
                       II_DayNumber := "ProdParam".DayNumber,
                       I_Melt := "ProdParam".Melt,
                       XS_MatCard := "STATUS_BSN2".MatCard[#CI_LastRow, 2],
                       XDI_PartID := #SDIPartID,
                       ENO => #_w22);
   IF #_w22 THEN "HMI_CMD_BSN2".Commands.MTS_Command.SetParts."22" := FALSE; END_IF;
   "MTS_CreateNewPart"(EN := "HMI_CMD_BSN2".Commands.MTS_Command.SetParts."23",
                       II_PartType := #SI_PartType,
                       II_DayNumber := "ProdParam".DayNumber,
                       I_Melt := "ProdParam".Melt,
                       XS_MatCard := "STATUS_BSN2".MatCard[#CI_LastRow, 3],
                       XDI_PartID := #SDIPartID,
                       ENO => #_w23);
   IF #_w23 THEN "HMI_CMD_BSN2".Commands.MTS_Command.SetParts."23" := FALSE; END_IF;
   "MTS_CreateNewPart"(EN := "HMI_CMD_BSN2".Commands.MTS_Command.SetParts."24",
                       II_PartType := #SI_PartType,
                       II_DayNumber := "ProdParam".DayNumber,
                       I_Melt := "ProdParam".Melt,
                       XS_MatCard := "STATUS_BSN2".MatCard[#CI_LastRow, 4],
                       XDI_PartID := #SDIPartID,
                       ENO => #_w24);
   IF #_w24 THEN "HMI_CMD_BSN2".Commands.MTS_Command.SetParts."24" := FALSE; END_IF;
   "MTS_CreateNewPart"(EN := "HMI_CMD_BSN2".Commands.MTS_Command.SetParts."25",
                       II_PartType := #SI_PartType,
                       II_DayNumber := "ProdParam".DayNumber,
                       I_Melt := "ProdParam".Melt,
                       XS_MatCard := "STATUS_BSN2".MatCard[#CI_LastRow, 5],
                       XDI_PartID := #SDIPartID,
                       ENO => #_w25);
   IF #_w25 THEN "HMI_CMD_BSN2".Commands.MTS_Command.SetParts."25" := FALSE; END_IF;
   "MTS_MapFill"(EN := "HMI_CMD_BSN2".Commands.MTS_Command.SetMap,
                 II_PartType := #SI_PartType,
                 X_Map := "STATUS_BSN2".MatCard,
                 ENO => #_w26);
   IF #_w26 THEN "HMI_CMD_BSN2".Commands.MTS_Command.SetMap := FALSE; END_IF;
END_REGION

REGION Network 17: Clear positions in map
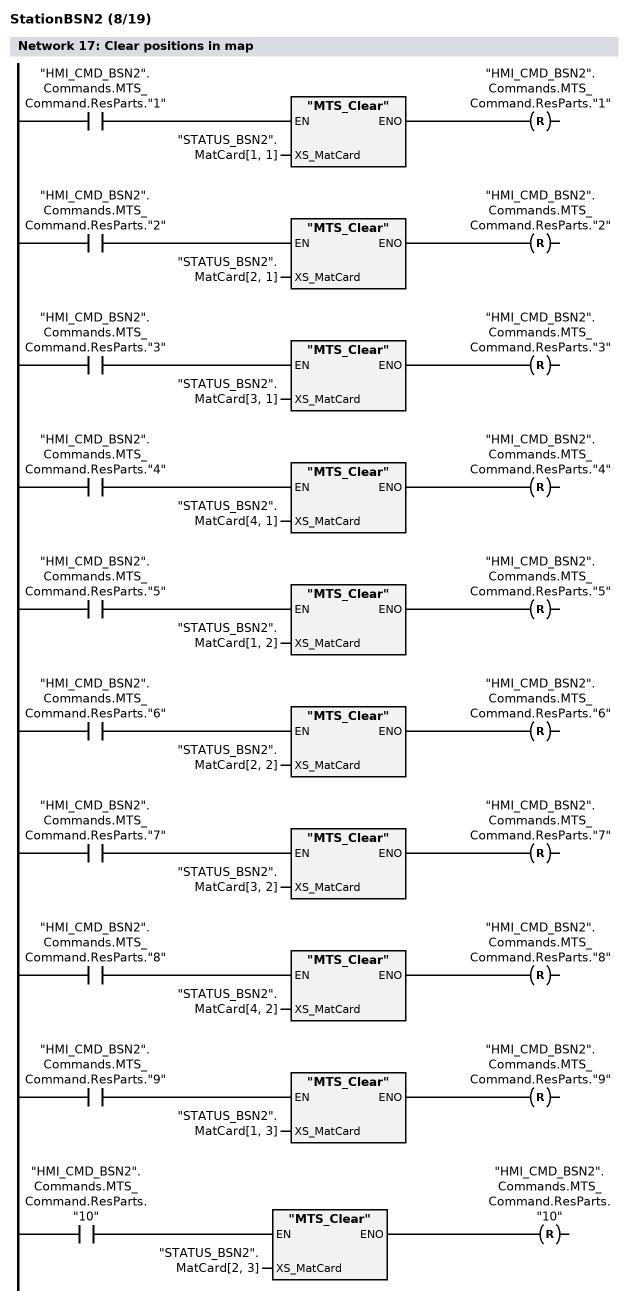
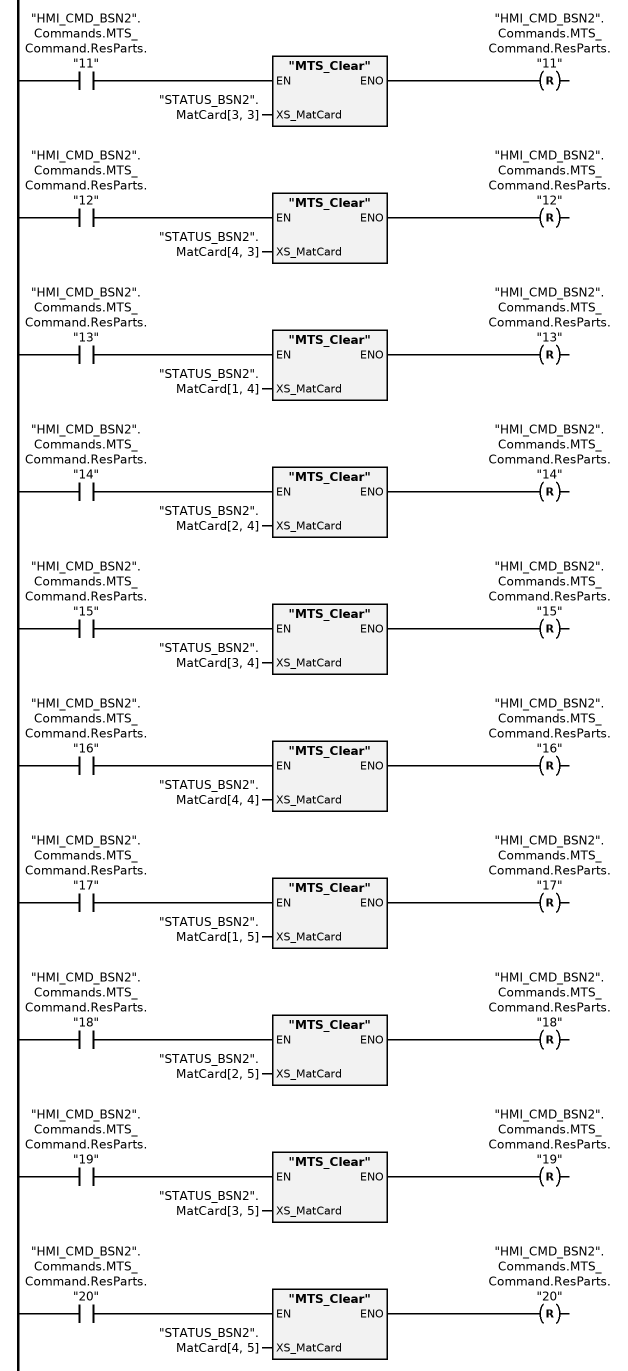
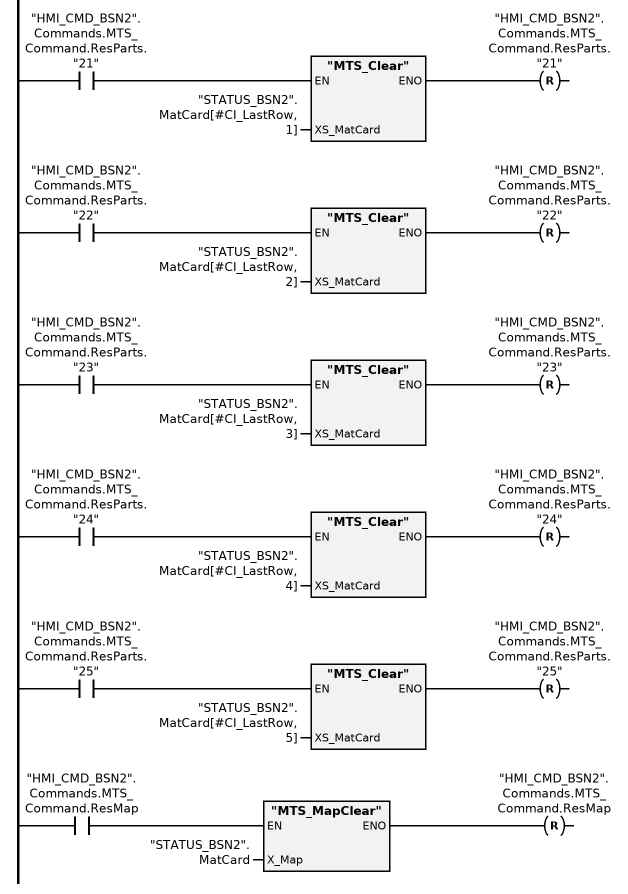
   RUNG wire#powerrail
      Contact( "HMI_CMD_BSN2".Commands.MTS_Command.ResParts."1" )
      "MTS_Clear"(XS_MatCard := "STATUS_BSN2".MatCard[1, 1])
      R_Coil( "HMI_CMD_BSN2".Commands.MTS_Command.ResParts."1" )
   END_RUNG
   RUNG wire#powerrail
      Contact( "HMI_CMD_BSN2".Commands.MTS_Command.ResParts."2" )
      "MTS_Clear"(XS_MatCard := "STATUS_BSN2".MatCard[2, 1])
      R_Coil( "HMI_CMD_BSN2".Commands.MTS_Command.ResParts."2" )
   END_RUNG
   RUNG wire#powerrail
      Contact( "HMI_CMD_BSN2".Commands.MTS_Command.ResParts."3" )
      "MTS_Clear"(XS_MatCard := "STATUS_BSN2".MatCard[3, 1])
      R_Coil( "HMI_CMD_BSN2".Commands.MTS_Command.ResParts."3" )
   END_RUNG
   RUNG wire#powerrail
      Contact( "HMI_CMD_BSN2".Commands.MTS_Command.ResParts."4" )
      "MTS_Clear"(XS_MatCard := "STATUS_BSN2".MatCard[4, 1])
      R_Coil( "HMI_CMD_BSN2".Commands.MTS_Command.ResParts."4" )
   END_RUNG
   RUNG wire#powerrail
      Contact( "HMI_CMD_BSN2".Commands.MTS_Command.ResParts."5" )
      "MTS_Clear"(XS_MatCard := "STATUS_BSN2".MatCard[1, 2])
      R_Coil( "HMI_CMD_BSN2".Commands.MTS_Command.ResParts."5" )
   END_RUNG
   RUNG wire#powerrail
      Contact( "HMI_CMD_BSN2".Commands.MTS_Command.ResParts."6" )
      "MTS_Clear"(XS_MatCard := "STATUS_BSN2".MatCard[2, 2])
      R_Coil( "HMI_CMD_BSN2".Commands.MTS_Command.ResParts."6" )
   END_RUNG
   RUNG wire#powerrail
      Contact( "HMI_CMD_BSN2".Commands.MTS_Command.ResParts."7" )
      "MTS_Clear"(XS_MatCard := "STATUS_BSN2".MatCard[3, 2])
      R_Coil( "HMI_CMD_BSN2".Commands.MTS_Command.ResParts."7" )
   END_RUNG
   RUNG wire#powerrail
      Contact( "HMI_CMD_BSN2".Commands.MTS_Command.ResParts."8" )
      "MTS_Clear"(XS_MatCard := "STATUS_BSN2".MatCard[4, 2])
      R_Coil( "HMI_CMD_BSN2".Commands.MTS_Command.ResParts."8" )
   END_RUNG
   RUNG wire#powerrail
      Contact( "HMI_CMD_BSN2".Commands.MTS_Command.ResParts."9" )
      "MTS_Clear"(XS_MatCard := "STATUS_BSN2".MatCard[1, 3])
      R_Coil( "HMI_CMD_BSN2".Commands.MTS_Command.ResParts."9" )
   END_RUNG
   RUNG wire#powerrail
      Contact( "HMI_CMD_BSN2".Commands.MTS_Command.ResParts."10" )
      "MTS_Clear"(XS_MatCard := "STATUS_BSN2".MatCard[2, 3])
      R_Coil( "HMI_CMD_BSN2".Commands.MTS_Command.ResParts."10" )
   END_RUNG
   RUNG wire#powerrail
      Contact( "HMI_CMD_BSN2".Commands.MTS_Command.ResParts."11" )
      "MTS_Clear"(XS_MatCard := "STATUS_BSN2".MatCard[3, 3])
      R_Coil( "HMI_CMD_BSN2".Commands.MTS_Command.ResParts."11" )
   END_RUNG
   RUNG wire#powerrail
      Contact( "HMI_CMD_BSN2".Commands.MTS_Command.ResParts."12" )
      "MTS_Clear"(XS_MatCard := "STATUS_BSN2".MatCard[4, 3])
      R_Coil( "HMI_CMD_BSN2".Commands.MTS_Command.ResParts."12" )
   END_RUNG
   RUNG wire#powerrail
      Contact( "HMI_CMD_BSN2".Commands.MTS_Command.ResParts."13" )
      "MTS_Clear"(XS_MatCard := "STATUS_BSN2".MatCard[1, 4])
      R_Coil( "HMI_CMD_BSN2".Commands.MTS_Command.ResParts."13" )
   END_RUNG
   RUNG wire#powerrail
      Contact( "HMI_CMD_BSN2".Commands.MTS_Command.ResParts."14" )
      "MTS_Clear"(XS_MatCard := "STATUS_BSN2".MatCard[2, 4])
      R_Coil( "HMI_CMD_BSN2".Commands.MTS_Command.ResParts."14" )
   END_RUNG
   RUNG wire#powerrail
      Contact( "HMI_CMD_BSN2".Commands.MTS_Command.ResParts."15" )
      "MTS_Clear"(XS_MatCard := "STATUS_BSN2".MatCard[3, 4])
      R_Coil( "HMI_CMD_BSN2".Commands.MTS_Command.ResParts."15" )
   END_RUNG
   RUNG wire#powerrail
      Contact( "HMI_CMD_BSN2".Commands.MTS_Command.ResParts."16" )
      "MTS_Clear"(XS_MatCard := "STATUS_BSN2".MatCard[4, 4])
      R_Coil( "HMI_CMD_BSN2".Commands.MTS_Command.ResParts."16" )
   END_RUNG
   RUNG wire#powerrail
      Contact( "HMI_CMD_BSN2".Commands.MTS_Command.ResParts."17" )
      "MTS_Clear"(XS_MatCard := "STATUS_BSN2".MatCard[1, 5])
      R_Coil( "HMI_CMD_BSN2".Commands.MTS_Command.ResParts."17" )
   END_RUNG
   RUNG wire#powerrail
      Contact( "HMI_CMD_BSN2".Commands.MTS_Command.ResParts."18" )
      "MTS_Clear"(XS_MatCard := "STATUS_BSN2".MatCard[2, 5])
      R_Coil( "HMI_CMD_BSN2".Commands.MTS_Command.ResParts."18" )
   END_RUNG
   RUNG wire#powerrail
      Contact( "HMI_CMD_BSN2".Commands.MTS_Command.ResParts."19" )
      "MTS_Clear"(XS_MatCard := "STATUS_BSN2".MatCard[3, 5])
      R_Coil( "HMI_CMD_BSN2".Commands.MTS_Command.ResParts."19" )
   END_RUNG
   RUNG wire#powerrail
      Contact( "HMI_CMD_BSN2".Commands.MTS_Command.ResParts."20" )
      "MTS_Clear"(XS_MatCard := "STATUS_BSN2".MatCard[4, 5])
      R_Coil( "HMI_CMD_BSN2".Commands.MTS_Command.ResParts."20" )
   END_RUNG
   RUNG wire#powerrail
      Contact( "HMI_CMD_BSN2".Commands.MTS_Command.ResParts."21" )
      "MTS_Clear"(XS_MatCard := "STATUS_BSN2".MatCard[#CI_LastRow, 1])
      R_Coil( "HMI_CMD_BSN2".Commands.MTS_Command.ResParts."21" )
   END_RUNG
   RUNG wire#powerrail
      Contact( "HMI_CMD_BSN2".Commands.MTS_Command.ResParts."22" )
      "MTS_Clear"(XS_MatCard := "STATUS_BSN2".MatCard[#CI_LastRow, 2])
      R_Coil( "HMI_CMD_BSN2".Commands.MTS_Command.ResParts."22" )
   END_RUNG
   RUNG wire#powerrail
      Contact( "HMI_CMD_BSN2".Commands.MTS_Command.ResParts."23" )
      "MTS_Clear"(XS_MatCard := "STATUS_BSN2".MatCard[#CI_LastRow, 3])
      R_Coil( "HMI_CMD_BSN2".Commands.MTS_Command.ResParts."23" )
   END_RUNG
   RUNG wire#powerrail
      Contact( "HMI_CMD_BSN2".Commands.MTS_Command.ResParts."24" )
      "MTS_Clear"(XS_MatCard := "STATUS_BSN2".MatCard[#CI_LastRow, 4])
      R_Coil( "HMI_CMD_BSN2".Commands.MTS_Command.ResParts."24" )
   END_RUNG
   RUNG wire#powerrail
      Contact( "HMI_CMD_BSN2".Commands.MTS_Command.ResParts."25" )
      "MTS_Clear"(XS_MatCard := "STATUS_BSN2".MatCard[#CI_LastRow, 5])
      R_Coil( "HMI_CMD_BSN2".Commands.MTS_Command.ResParts."25" )
   END_RUNG
   RUNG wire#powerrail
      Contact( "HMI_CMD_BSN2".Commands.MTS_Command.ResMap )
      "MTS_MapClear"(X_Map := "STATUS_BSN2".MatCard)
      R_Coil( "HMI_CMD_BSN2".Commands.MTS_Command.ResMap )
   END_RUNG
   // the same network as SCL:
   "MTS_Clear"(EN := "HMI_CMD_BSN2".Commands.MTS_Command.ResParts."1",
               XS_MatCard := "STATUS_BSN2".MatCard[1, 1],
               ENO => #_w1);
   IF #_w1 THEN "HMI_CMD_BSN2".Commands.MTS_Command.ResParts."1" := FALSE; END_IF;
   "MTS_Clear"(EN := "HMI_CMD_BSN2".Commands.MTS_Command.ResParts."2",
               XS_MatCard := "STATUS_BSN2".MatCard[2, 1],
               ENO => #_w2);
   IF #_w2 THEN "HMI_CMD_BSN2".Commands.MTS_Command.ResParts."2" := FALSE; END_IF;
   "MTS_Clear"(EN := "HMI_CMD_BSN2".Commands.MTS_Command.ResParts."3",
               XS_MatCard := "STATUS_BSN2".MatCard[3, 1],
               ENO => #_w3);
   IF #_w3 THEN "HMI_CMD_BSN2".Commands.MTS_Command.ResParts."3" := FALSE; END_IF;
   "MTS_Clear"(EN := "HMI_CMD_BSN2".Commands.MTS_Command.ResParts."4",
               XS_MatCard := "STATUS_BSN2".MatCard[4, 1],
               ENO => #_w4);
   IF #_w4 THEN "HMI_CMD_BSN2".Commands.MTS_Command.ResParts."4" := FALSE; END_IF;
   "MTS_Clear"(EN := "HMI_CMD_BSN2".Commands.MTS_Command.ResParts."5",
               XS_MatCard := "STATUS_BSN2".MatCard[1, 2],
               ENO => #_w5);
   IF #_w5 THEN "HMI_CMD_BSN2".Commands.MTS_Command.ResParts."5" := FALSE; END_IF;
   "MTS_Clear"(EN := "HMI_CMD_BSN2".Commands.MTS_Command.ResParts."6",
               XS_MatCard := "STATUS_BSN2".MatCard[2, 2],
               ENO => #_w6);
   IF #_w6 THEN "HMI_CMD_BSN2".Commands.MTS_Command.ResParts."6" := FALSE; END_IF;
   "MTS_Clear"(EN := "HMI_CMD_BSN2".Commands.MTS_Command.ResParts."7",
               XS_MatCard := "STATUS_BSN2".MatCard[3, 2],
               ENO => #_w7);
   IF #_w7 THEN "HMI_CMD_BSN2".Commands.MTS_Command.ResParts."7" := FALSE; END_IF;
   "MTS_Clear"(EN := "HMI_CMD_BSN2".Commands.MTS_Command.ResParts."8",
               XS_MatCard := "STATUS_BSN2".MatCard[4, 2],
               ENO => #_w8);
   IF #_w8 THEN "HMI_CMD_BSN2".Commands.MTS_Command.ResParts."8" := FALSE; END_IF;
   "MTS_Clear"(EN := "HMI_CMD_BSN2".Commands.MTS_Command.ResParts."9",
               XS_MatCard := "STATUS_BSN2".MatCard[1, 3],
               ENO => #_w9);
   IF #_w9 THEN "HMI_CMD_BSN2".Commands.MTS_Command.ResParts."9" := FALSE; END_IF;
   "MTS_Clear"(EN := "HMI_CMD_BSN2".Commands.MTS_Command.ResParts."10",
               XS_MatCard := "STATUS_BSN2".MatCard[2, 3],
               ENO => #_w10);
   IF #_w10 THEN "HMI_CMD_BSN2".Commands.MTS_Command.ResParts."10" := FALSE; END_IF;
   "MTS_Clear"(EN := "HMI_CMD_BSN2".Commands.MTS_Command.ResParts."11",
               XS_MatCard := "STATUS_BSN2".MatCard[3, 3],
               ENO => #_w11);
   IF #_w11 THEN "HMI_CMD_BSN2".Commands.MTS_Command.ResParts."11" := FALSE; END_IF;
   "MTS_Clear"(EN := "HMI_CMD_BSN2".Commands.MTS_Command.ResParts."12",
               XS_MatCard := "STATUS_BSN2".MatCard[4, 3],
               ENO => #_w12);
   IF #_w12 THEN "HMI_CMD_BSN2".Commands.MTS_Command.ResParts."12" := FALSE; END_IF;
   "MTS_Clear"(EN := "HMI_CMD_BSN2".Commands.MTS_Command.ResParts."13",
               XS_MatCard := "STATUS_BSN2".MatCard[1, 4],
               ENO => #_w13);
   IF #_w13 THEN "HMI_CMD_BSN2".Commands.MTS_Command.ResParts."13" := FALSE; END_IF;
   "MTS_Clear"(EN := "HMI_CMD_BSN2".Commands.MTS_Command.ResParts."14",
               XS_MatCard := "STATUS_BSN2".MatCard[2, 4],
               ENO => #_w14);
   IF #_w14 THEN "HMI_CMD_BSN2".Commands.MTS_Command.ResParts."14" := FALSE; END_IF;
   "MTS_Clear"(EN := "HMI_CMD_BSN2".Commands.MTS_Command.ResParts."15",
               XS_MatCard := "STATUS_BSN2".MatCard[3, 4],
               ENO => #_w15);
   IF #_w15 THEN "HMI_CMD_BSN2".Commands.MTS_Command.ResParts."15" := FALSE; END_IF;
   "MTS_Clear"(EN := "HMI_CMD_BSN2".Commands.MTS_Command.ResParts."16",
               XS_MatCard := "STATUS_BSN2".MatCard[4, 4],
               ENO => #_w16);
   IF #_w16 THEN "HMI_CMD_BSN2".Commands.MTS_Command.ResParts."16" := FALSE; END_IF;
   "MTS_Clear"(EN := "HMI_CMD_BSN2".Commands.MTS_Command.ResParts."17",
               XS_MatCard := "STATUS_BSN2".MatCard[1, 5],
               ENO => #_w17);
   IF #_w17 THEN "HMI_CMD_BSN2".Commands.MTS_Command.ResParts."17" := FALSE; END_IF;
   "MTS_Clear"(EN := "HMI_CMD_BSN2".Commands.MTS_Command.ResParts."18",
               XS_MatCard := "STATUS_BSN2".MatCard[2, 5],
               ENO => #_w18);
   IF #_w18 THEN "HMI_CMD_BSN2".Commands.MTS_Command.ResParts."18" := FALSE; END_IF;
   "MTS_Clear"(EN := "HMI_CMD_BSN2".Commands.MTS_Command.ResParts."19",
               XS_MatCard := "STATUS_BSN2".MatCard[3, 5],
               ENO => #_w19);
   IF #_w19 THEN "HMI_CMD_BSN2".Commands.MTS_Command.ResParts."19" := FALSE; END_IF;
   "MTS_Clear"(EN := "HMI_CMD_BSN2".Commands.MTS_Command.ResParts."20",
               XS_MatCard := "STATUS_BSN2".MatCard[4, 5],
               ENO => #_w20);
   IF #_w20 THEN "HMI_CMD_BSN2".Commands.MTS_Command.ResParts."20" := FALSE; END_IF;
   "MTS_Clear"(EN := "HMI_CMD_BSN2".Commands.MTS_Command.ResParts."21",
               XS_MatCard := "STATUS_BSN2".MatCard[#CI_LastRow, 1],
               ENO => #_w21);
   IF #_w21 THEN "HMI_CMD_BSN2".Commands.MTS_Command.ResParts."21" := FALSE; END_IF;
   "MTS_Clear"(EN := "HMI_CMD_BSN2".Commands.MTS_Command.ResParts."22",
               XS_MatCard := "STATUS_BSN2".MatCard[#CI_LastRow, 2],
               ENO => #_w22);
   IF #_w22 THEN "HMI_CMD_BSN2".Commands.MTS_Command.ResParts."22" := FALSE; END_IF;
   "MTS_Clear"(EN := "HMI_CMD_BSN2".Commands.MTS_Command.ResParts."23",
               XS_MatCard := "STATUS_BSN2".MatCard[#CI_LastRow, 3],
               ENO => #_w23);
   IF #_w23 THEN "HMI_CMD_BSN2".Commands.MTS_Command.ResParts."23" := FALSE; END_IF;
   "MTS_Clear"(EN := "HMI_CMD_BSN2".Commands.MTS_Command.ResParts."24",
               XS_MatCard := "STATUS_BSN2".MatCard[#CI_LastRow, 4],
               ENO => #_w24);
   IF #_w24 THEN "HMI_CMD_BSN2".Commands.MTS_Command.ResParts."24" := FALSE; END_IF;
   "MTS_Clear"(EN := "HMI_CMD_BSN2".Commands.MTS_Command.ResParts."25",
               XS_MatCard := "STATUS_BSN2".MatCard[#CI_LastRow, 5],
               ENO => #_w25);
   IF #_w25 THEN "HMI_CMD_BSN2".Commands.MTS_Command.ResParts."25" := FALSE; END_IF;
   "MTS_MapClear"(EN := "HMI_CMD_BSN2".Commands.MTS_Command.ResMap,
                  X_Map := "STATUS_BSN2".MatCard,
                  ENO => #_w26);
   IF #_w26 THEN "HMI_CMD_BSN2".Commands.MTS_Command.ResMap := FALSE; END_IF;
END_REGION

REGION Network 18: Clear positions on output conveyor
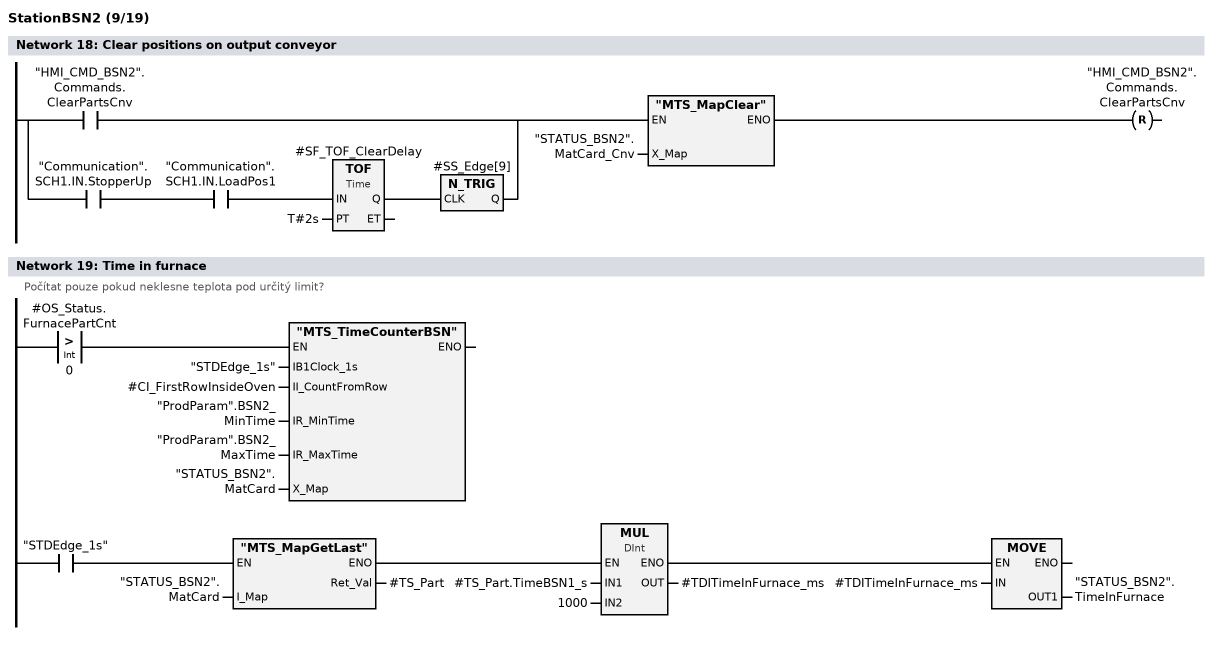
   RUNG wire#powerrail
      Contact( "HMI_CMD_BSN2".Commands.ClearPartsCnv )
      wire#w1
      "MTS_MapClear"(X_Map := "STATUS_BSN2".MatCard_Cnv)
      R_Coil( "HMI_CMD_BSN2".Commands.ClearPartsCnv )
   END_RUNG
   RUNG wire#powerrail
      Contact( "Communication".SCH1.IN.StopperUp )
      Contact( "Communication".SCH1.IN.LoadPos1 )
      { S7_Templates := "time_type := Time" } #SF_TOF_ClearDelay.TOF(pt := T#2s, et =>)
      N_Trig( #SS_Edge[9] )
   END_RUNG wire#w1
   // the same network as SCL:
   #SF_TOF_ClearDelay(IN := "Communication".SCH1.IN.StopperUp AND "Communication".SCH1.IN.LoadPos1, PT := T#2s);   // TOF
   #_w1 := NOT #SF_TOF_ClearDelay.Q AND #SS_Edge[9];   // falling edge
   #SS_Edge[9] := #SF_TOF_ClearDelay.Q;
   "MTS_MapClear"(EN := "HMI_CMD_BSN2".Commands.ClearPartsCnv OR #_w1,
                  X_Map := "STATUS_BSN2".MatCard_Cnv,
                  ENO => #_w2);
   IF #_w2 THEN "HMI_CMD_BSN2".Commands.ClearPartsCnv := FALSE; END_IF;
END_REGION

REGION Network 19: Time in furnace
   // Počítat pouze pokud neklesne teplota pod určitý limit?
   RUNG wire#powerrail
      { S7_Templates := "SrcType := Int" } GT_Contact(in1 := #OS_Status.FurnacePartCnt, in2 := 0)
      "MTS_TimeCounterBSN"(IB1Clock_1s := "STDEdge_1s", II_CountFromRow := #CI_FirstRowInsideOven, IR_MinTime := "ProdParam".BSN2_MinTime, IR_MaxTime := "ProdParam".BSN2_MaxTime, X_Map := "STATUS_BSN2".MatCard)
   END_RUNG
   RUNG wire#powerrail
      Contact( "STDEdge_1s" )
      "MTS_MapGetLast"(I_Map := "STATUS_BSN2".MatCard, Ret_Val => #TS_Part)
      { S7_Templates := "SrcType := DInt"; S7_GenerateENO := "TRUE" } Mul(in1 := #TS_Part.TimeBSN1_s, in2 := 1000, out => #TDITimeInFurnace_ms)
      Move(in := #TDITimeInFurnace_ms, out1 => "STATUS_BSN2".TimeInFurnace)
   END_RUNG
   // the same network as SCL:
   // ENO of a box is taken as its EN; it also drops when the box reports an error
   IF #OS_Status.FurnacePartCnt > 0 THEN
       "MTS_TimeCounterBSN"(IB1Clock_1s := "STDEdge_1s",
                            II_CountFromRow := #CI_FirstRowInsideOven,
                            IR_MinTime := "ProdParam".BSN2_MinTime,
                            IR_MaxTime := "ProdParam".BSN2_MaxTime,
                            X_Map := "STATUS_BSN2".MatCard);
   END_IF;
   #TS_Part := "MTS_MapGetLast"(EN := "STDEdge_1s", I_Map := "STATUS_BSN2".MatCard, ENO => #_w1);
   IF #_w1 THEN
       #TDITimeInFurnace_ms := #TS_Part.TimeBSN1_s * 1000;
       "STATUS_BSN2".TimeInFurnace := #TDITimeInFurnace_ms;
   END_IF;
END_REGION

REGION Network 20: Time on output conveyor
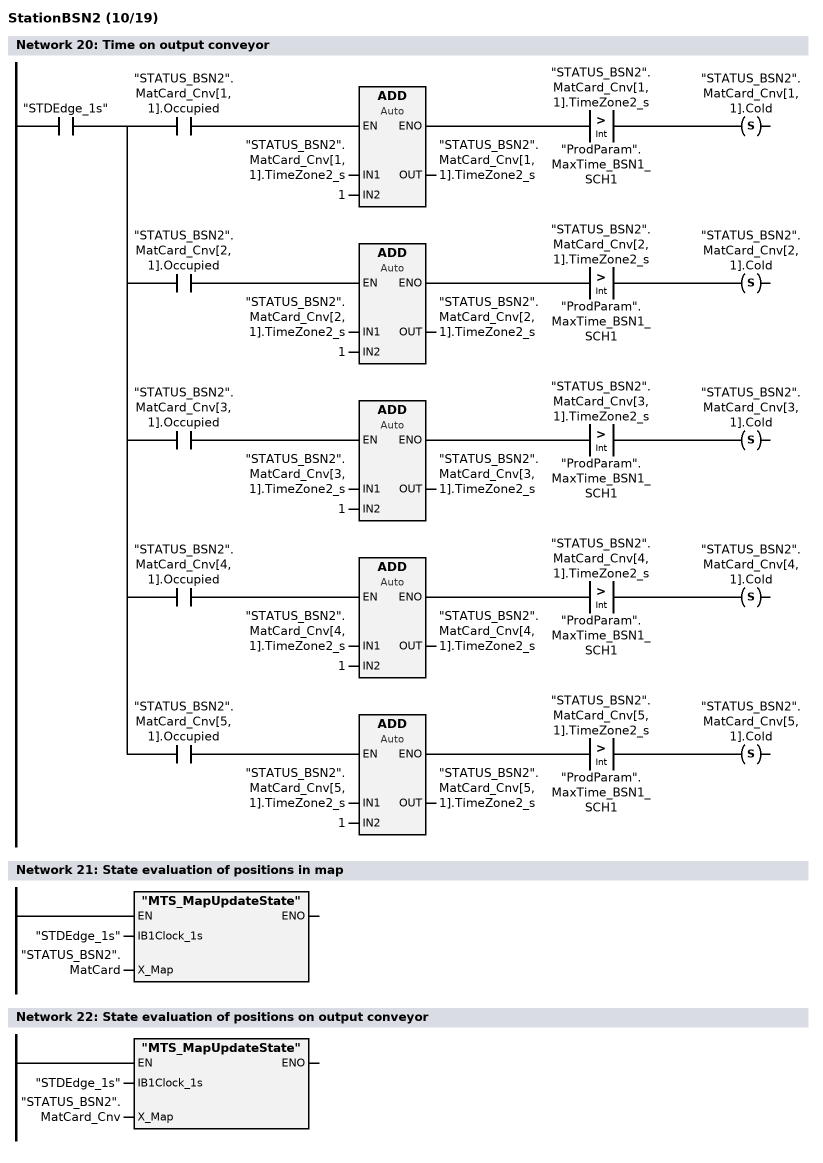
   RUNG wire#powerrail
      Contact( "STDEdge_1s" )
      wire#w1
      Contact( "STATUS_BSN2".MatCard_Cnv[1, 1].Occupied )
      Add(in1 := "STATUS_BSN2".MatCard_Cnv[1, 1].TimeZone2_s, in2 := 1, out => "STATUS_BSN2".MatCard_Cnv[1, 1].TimeZone2_s)
      { S7_Templates := "SrcType := Int" } GT_Contact(in1 := "STATUS_BSN2".MatCard_Cnv[1, 1].TimeZone2_s, in2 := "ProdParam".MaxTime_BSN1_SCH1)
      S_Coil( "STATUS_BSN2".MatCard_Cnv[1, 1].Cold )
   END_RUNG
   RUNG wire#w1
      Contact( "STATUS_BSN2".MatCard_Cnv[2, 1].Occupied )
      Add(in1 := "STATUS_BSN2".MatCard_Cnv[2, 1].TimeZone2_s, in2 := 1, out => "STATUS_BSN2".MatCard_Cnv[2, 1].TimeZone2_s)
      { S7_Templates := "SrcType := Int" } GT_Contact(in1 := "STATUS_BSN2".MatCard_Cnv[2, 1].TimeZone2_s, in2 := "ProdParam".MaxTime_BSN1_SCH1)
      S_Coil( "STATUS_BSN2".MatCard_Cnv[2, 1].Cold )
   END_RUNG
   RUNG wire#w1
      Contact( "STATUS_BSN2".MatCard_Cnv[3, 1].Occupied )
      Add(in1 := "STATUS_BSN2".MatCard_Cnv[3, 1].TimeZone2_s, in2 := 1, out => "STATUS_BSN2".MatCard_Cnv[3, 1].TimeZone2_s)
      { S7_Templates := "SrcType := Int" } GT_Contact(in1 := "STATUS_BSN2".MatCard_Cnv[3, 1].TimeZone2_s, in2 := "ProdParam".MaxTime_BSN1_SCH1)
      S_Coil( "STATUS_BSN2".MatCard_Cnv[3, 1].Cold )
   END_RUNG
   RUNG wire#w1
      Contact( "STATUS_BSN2".MatCard_Cnv[4, 1].Occupied )
      Add(in1 := "STATUS_BSN2".MatCard_Cnv[4, 1].TimeZone2_s, in2 := 1, out => "STATUS_BSN2".MatCard_Cnv[4, 1].TimeZone2_s)
      { S7_Templates := "SrcType := Int" } GT_Contact(in1 := "STATUS_BSN2".MatCard_Cnv[4, 1].TimeZone2_s, in2 := "ProdParam".MaxTime_BSN1_SCH1)
      S_Coil( "STATUS_BSN2".MatCard_Cnv[4, 1].Cold )
   END_RUNG
   RUNG wire#w1
      Contact( "STATUS_BSN2".MatCard_Cnv[5, 1].Occupied )
      Add(in1 := "STATUS_BSN2".MatCard_Cnv[5, 1].TimeZone2_s, in2 := 1, out => "STATUS_BSN2".MatCard_Cnv[5, 1].TimeZone2_s)
      { S7_Templates := "SrcType := Int" } GT_Contact(in1 := "STATUS_BSN2".MatCard_Cnv[5, 1].TimeZone2_s, in2 := "ProdParam".MaxTime_BSN1_SCH1)
      S_Coil( "STATUS_BSN2".MatCard_Cnv[5, 1].Cold )
   END_RUNG
   // the same network as SCL:
   #_w1 := "STDEdge_1s" AND "STATUS_BSN2".MatCard_Cnv[1, 1].Occupied;
   IF #_w1 THEN
       "STATUS_BSN2".MatCard_Cnv[1, 1].TimeZone2_s := "STATUS_BSN2".MatCard_Cnv[1, 1].TimeZone2_s + 1;
   END_IF;
   IF #_w1 AND ("STATUS_BSN2".MatCard_Cnv[1, 1].TimeZone2_s > "ProdParam".MaxTime_BSN1_SCH1) THEN
       "STATUS_BSN2".MatCard_Cnv[1, 1].Cold := TRUE;
   END_IF;
   #_w2 := "STDEdge_1s" AND "STATUS_BSN2".MatCard_Cnv[2, 1].Occupied;
   IF #_w2 THEN
       "STATUS_BSN2".MatCard_Cnv[2, 1].TimeZone2_s := "STATUS_BSN2".MatCard_Cnv[2, 1].TimeZone2_s + 1;
   END_IF;
   IF #_w2 AND ("STATUS_BSN2".MatCard_Cnv[2, 1].TimeZone2_s > "ProdParam".MaxTime_BSN1_SCH1) THEN
       "STATUS_BSN2".MatCard_Cnv[2, 1].Cold := TRUE;
   END_IF;
   #_w3 := "STDEdge_1s" AND "STATUS_BSN2".MatCard_Cnv[3, 1].Occupied;
   IF #_w3 THEN
       "STATUS_BSN2".MatCard_Cnv[3, 1].TimeZone2_s := "STATUS_BSN2".MatCard_Cnv[3, 1].TimeZone2_s + 1;
   END_IF;
   IF #_w3 AND ("STATUS_BSN2".MatCard_Cnv[3, 1].TimeZone2_s > "ProdParam".MaxTime_BSN1_SCH1) THEN
       "STATUS_BSN2".MatCard_Cnv[3, 1].Cold := TRUE;
   END_IF;
   #_w4 := "STDEdge_1s" AND "STATUS_BSN2".MatCard_Cnv[4, 1].Occupied;
   IF #_w4 THEN
       "STATUS_BSN2".MatCard_Cnv[4, 1].TimeZone2_s := "STATUS_BSN2".MatCard_Cnv[4, 1].TimeZone2_s + 1;
   END_IF;
   IF #_w4 AND ("STATUS_BSN2".MatCard_Cnv[4, 1].TimeZone2_s > "ProdParam".MaxTime_BSN1_SCH1) THEN
       "STATUS_BSN2".MatCard_Cnv[4, 1].Cold := TRUE;
   END_IF;
   #_w5 := "STDEdge_1s" AND "STATUS_BSN2".MatCard_Cnv[5, 1].Occupied;
   IF #_w5 THEN
       "STATUS_BSN2".MatCard_Cnv[5, 1].TimeZone2_s := "STATUS_BSN2".MatCard_Cnv[5, 1].TimeZone2_s + 1;
   END_IF;
   IF #_w5 AND ("STATUS_BSN2".MatCard_Cnv[5, 1].TimeZone2_s > "ProdParam".MaxTime_BSN1_SCH1) THEN
       "STATUS_BSN2".MatCard_Cnv[5, 1].Cold := TRUE;
   END_IF;
END_REGION

REGION Network 21: State evaluation of positions in map
   RUNG wire#powerrail
      "MTS_MapUpdateState"(IB1Clock_1s := "STDEdge_1s", X_Map := "STATUS_BSN2".MatCard)
   END_RUNG
   // the same network as SCL:
   "MTS_MapUpdateState"(IB1Clock_1s := "STDEdge_1s", X_Map := "STATUS_BSN2".MatCard);
END_REGION

REGION Network 22: State evaluation of positions on output conveyor
   RUNG wire#powerrail
      "MTS_MapUpdateState"(IB1Clock_1s := "STDEdge_1s", X_Map := "STATUS_BSN2".MatCard_Cnv)
   END_RUNG
   // the same network as SCL:
   "MTS_MapUpdateState"(IB1Clock_1s := "STDEdge_1s", X_Map := "STATUS_BSN2".MatCard_Cnv);
END_REGION

REGION Network 23: Data transfer: Map move
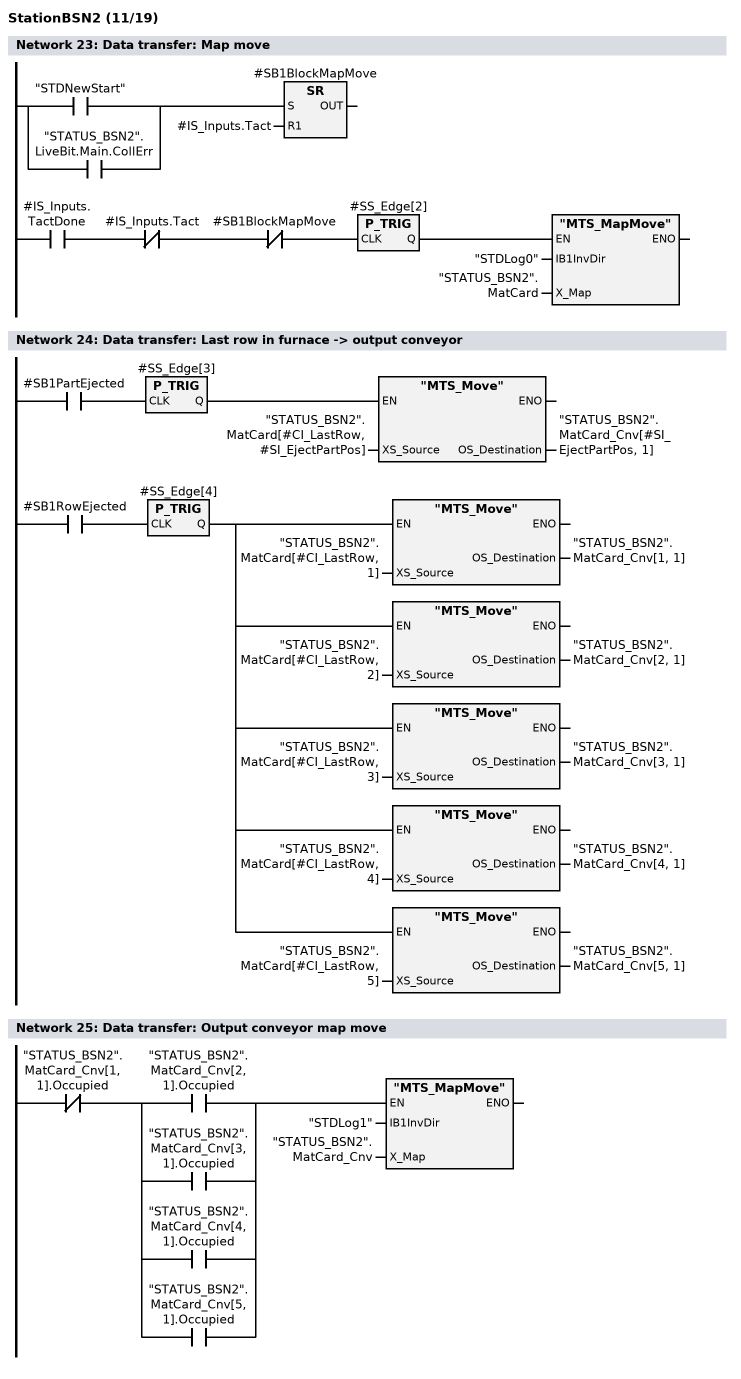
   RUNG wire#powerrail
      Contact( "STDNewStart" )
      wire#w1
      S_SR(operand := #SB1BlockMapMove, r1 := #IS_Inputs.Tact)
   END_RUNG
   RUNG wire#powerrail
      Contact( "STATUS_BSN2".LiveBit.Main.CollErr )
   END_RUNG wire#w1
   RUNG wire#powerrail
      Contact( #IS_Inputs.TactDone )
      I_Contact( #IS_Inputs.Tact )
      I_Contact( #SB1BlockMapMove )
      P_Trig( #SS_Edge[2] )
      "MTS_MapMove"(IB1InvDir := "STDLog0", X_Map := "STATUS_BSN2".MatCard)
   END_RUNG
   // the same network as SCL:
   IF "STDNewStart" OR "STATUS_BSN2".LiveBit.Main.CollErr THEN
       #SB1BlockMapMove := TRUE;   // SR flip-flop
   END_IF;
   IF #IS_Inputs.Tact THEN #SB1BlockMapMove := FALSE; END_IF;
   #_w1 := #IS_Inputs.TactDone AND NOT #IS_Inputs.Tact AND NOT #SB1BlockMapMove;
   #_w2 := #_w1 AND NOT #SS_Edge[2];   // rising edge
   #SS_Edge[2] := #_w1;
   IF #_w2 THEN "MTS_MapMove"(IB1InvDir := "STDLog0", X_Map := "STATUS_BSN2".MatCard); END_IF;
END_REGION

REGION Network 24: Data transfer: Last row in furnace -> output conveyor
   RUNG wire#powerrail
      Contact( #SB1PartEjected )
      P_Trig( #SS_Edge[3] )
      "MTS_Move"(XS_Source := "STATUS_BSN2".MatCard[#CI_LastRow, #SI_EjectPartPos], OS_Destination => "STATUS_BSN2".MatCard_Cnv[#SI_EjectPartPos, 1])
   END_RUNG
   RUNG wire#powerrail
      Contact( #SB1RowEjected )
      P_Trig( #SS_Edge[4] )
      wire#w1
      "MTS_Move"(XS_Source := "STATUS_BSN2".MatCard[#CI_LastRow, 1], OS_Destination => "STATUS_BSN2".MatCard_Cnv[1, 1])
   END_RUNG
   RUNG wire#w1
      "MTS_Move"(XS_Source := "STATUS_BSN2".MatCard[#CI_LastRow, 2], OS_Destination => "STATUS_BSN2".MatCard_Cnv[2, 1])
   END_RUNG
   RUNG wire#w1
      "MTS_Move"(XS_Source := "STATUS_BSN2".MatCard[#CI_LastRow, 3], OS_Destination => "STATUS_BSN2".MatCard_Cnv[3, 1])
   END_RUNG
   RUNG wire#w1
      "MTS_Move"(XS_Source := "STATUS_BSN2".MatCard[#CI_LastRow, 4], OS_Destination => "STATUS_BSN2".MatCard_Cnv[4, 1])
   END_RUNG
   RUNG wire#w1
      "MTS_Move"(XS_Source := "STATUS_BSN2".MatCard[#CI_LastRow, 5], OS_Destination => "STATUS_BSN2".MatCard_Cnv[5, 1])
   END_RUNG
   // the same network as SCL:
   #_w1 := #SB1PartEjected AND NOT #SS_Edge[3];   // rising edge
   #SS_Edge[3] := #SB1PartEjected;
   IF #_w1 THEN
       "MTS_Move"(XS_Source := "STATUS_BSN2".MatCard[#CI_LastRow, #SI_EjectPartPos],
                  OS_Destination => "STATUS_BSN2".MatCard_Cnv[#SI_EjectPartPos, 1]);
   END_IF;
   #_w2 := #SB1RowEjected AND NOT #SS_Edge[4];   // rising edge
   #SS_Edge[4] := #SB1RowEjected;
   IF #_w2 THEN
       "MTS_Move"(XS_Source := "STATUS_BSN2".MatCard[#CI_LastRow, 1],
                  OS_Destination => "STATUS_BSN2".MatCard_Cnv[1, 1]);
       "MTS_Move"(XS_Source := "STATUS_BSN2".MatCard[#CI_LastRow, 2],
                  OS_Destination => "STATUS_BSN2".MatCard_Cnv[2, 1]);
       "MTS_Move"(XS_Source := "STATUS_BSN2".MatCard[#CI_LastRow, 3],
                  OS_Destination => "STATUS_BSN2".MatCard_Cnv[3, 1]);
       "MTS_Move"(XS_Source := "STATUS_BSN2".MatCard[#CI_LastRow, 4],
                  OS_Destination => "STATUS_BSN2".MatCard_Cnv[4, 1]);
       "MTS_Move"(XS_Source := "STATUS_BSN2".MatCard[#CI_LastRow, 5],
                  OS_Destination => "STATUS_BSN2".MatCard_Cnv[5, 1]);
   END_IF;
END_REGION

REGION Network 25: Data transfer: Output conveyor map move
   RUNG wire#powerrail
      I_Contact( "STATUS_BSN2".MatCard_Cnv[1, 1].Occupied )
      wire#w1
      Contact( "STATUS_BSN2".MatCard_Cnv[2, 1].Occupied )
      wire#w2
      "MTS_MapMove"(IB1InvDir := "STDLog1", X_Map := "STATUS_BSN2".MatCard_Cnv)
   END_RUNG
   RUNG wire#w1
      Contact( "STATUS_BSN2".MatCard_Cnv[3, 1].Occupied )
   END_RUNG wire#w2
   RUNG wire#w1
      Contact( "STATUS_BSN2".MatCard_Cnv[4, 1].Occupied )
   END_RUNG wire#w2
   RUNG wire#w1
      Contact( "STATUS_BSN2".MatCard_Cnv[5, 1].Occupied )
   END_RUNG wire#w2
   // the same network as SCL:
   IF NOT "STATUS_BSN2".MatCard_Cnv[1, 1].Occupied AND ("STATUS_BSN2".MatCard_Cnv[2, 1].Occupied OR "STATUS_BSN2".MatCard_Cnv[3, 1].Occupied OR "STATUS_BSN2".MatCard_Cnv[4, 1].Occupied OR "STATUS_BSN2".MatCard_Cnv[5, 1].Occupied) THEN
       "MTS_MapMove"(IB1InvDir := "STDLog1", X_Map := "STATUS_BSN2".MatCard_Cnv);
   END_IF;
END_REGION

REGION Network 26: *************** Interface to furnace ***************
END_REGION

REGION Network 27: Live bit
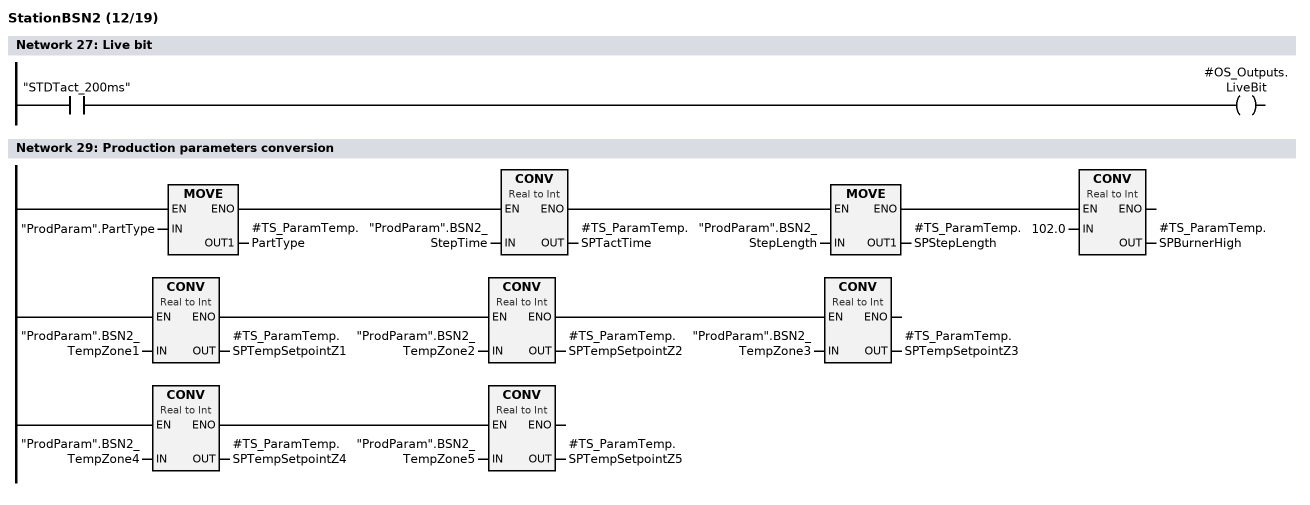
   RUNG wire#powerrail
      Contact( "STDTact_200ms" )
      Coil( #OS_Outputs.LiveBit )
   END_RUNG
   // the same network as SCL:
   #OS_Outputs.LiveBit := "STDTact_200ms";
END_REGION

REGION Network 28: ************** Production parameters ***************
END_REGION

REGION Network 29: Production parameters conversion
   RUNG wire#powerrail
      Move(in := "ProdParam".PartType, out1 => #TS_ParamTemp.PartType)
      { S7_Templates := "[SrcType := Real, DestType := Int]" } Convert(in := "ProdParam".BSN2_StepTime, out => #TS_ParamTemp.SPTactTime)
      Move(in := "ProdParam".BSN2_StepLength, out1 => #TS_ParamTemp.SPStepLength)
      { S7_Templates := "[SrcType := Real, DestType := Int]" } Convert(in := 102.0, out => #TS_ParamTemp.SPBurnerHigh)
   END_RUNG
   RUNG wire#powerrail
      { S7_Templates := "[SrcType := Real, DestType := Int]" } Convert(in := "ProdParam".BSN2_TempZone1, out => #TS_ParamTemp.SPTempSetpointZ1)
      { S7_Templates := "[SrcType := Real, DestType := Int]" } Convert(in := "ProdParam".BSN2_TempZone2, out => #TS_ParamTemp.SPTempSetpointZ2)
      { S7_Templates := "[SrcType := Real, DestType := Int]" } Convert(in := "ProdParam".BSN2_TempZone3, out => #TS_ParamTemp.SPTempSetpointZ3)
   END_RUNG
   RUNG wire#powerrail
      { S7_Templates := "[SrcType := Real, DestType := Int]" } Convert(in := "ProdParam".BSN2_TempZone4, out => #TS_ParamTemp.SPTempSetpointZ4)
      { S7_Templates := "[SrcType := Real, DestType := Int]" } Convert(in := "ProdParam".BSN2_TempZone5, out => #TS_ParamTemp.SPTempSetpointZ5)
   END_RUNG
   // the same network as SCL:
   #TS_ParamTemp.PartType := "ProdParam".PartType;
   #TS_ParamTemp.SPTactTime := REAL_TO_INT("ProdParam".BSN2_StepTime);
   #TS_ParamTemp.SPStepLength := "ProdParam".BSN2_StepLength;
   #TS_ParamTemp.SPBurnerHigh := REAL_TO_INT(102.0);
   #TS_ParamTemp.SPTempSetpointZ1 := REAL_TO_INT("ProdParam".BSN2_TempZone1);
   #TS_ParamTemp.SPTempSetpointZ2 := REAL_TO_INT("ProdParam".BSN2_TempZone2);
   #TS_ParamTemp.SPTempSetpointZ3 := REAL_TO_INT("ProdParam".BSN2_TempZone3);
   #TS_ParamTemp.SPTempSetpointZ4 := REAL_TO_INT("ProdParam".BSN2_TempZone4);
   #TS_ParamTemp.SPTempSetpointZ5 := REAL_TO_INT("ProdParam".BSN2_TempZone5);
END_REGION

REGION Network 30: Production parameter changed trigger
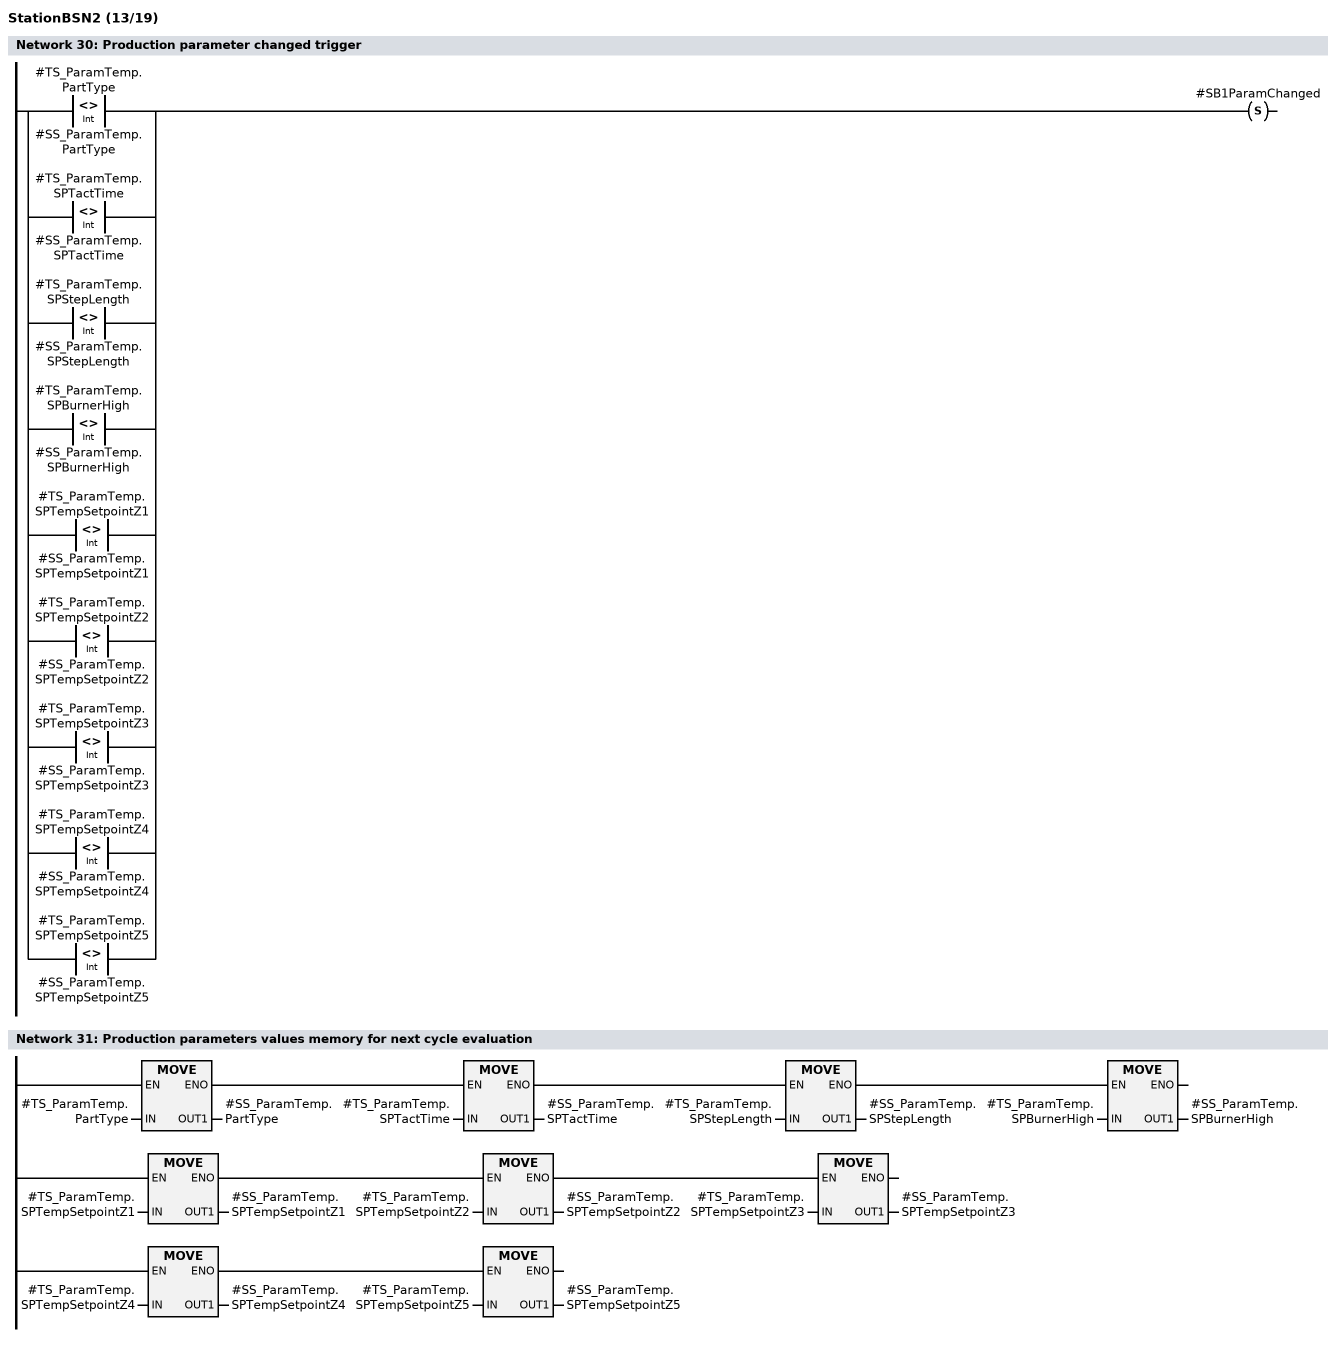
   RUNG wire#powerrail
      { S7_Templates := "SrcType := Int" } NE_Contact(in1 := #TS_ParamTemp.PartType, in2 := #SS_ParamTemp.PartType)
      wire#w1
      S_Coil( #SB1ParamChanged )
   END_RUNG
   RUNG wire#powerrail
      { S7_Templates := "SrcType := Int" } NE_Contact(in1 := #TS_ParamTemp.SPTactTime, in2 := #SS_ParamTemp.SPTactTime)
   END_RUNG wire#w1
   RUNG wire#powerrail
      { S7_Templates := "SrcType := Int" } NE_Contact(in1 := #TS_ParamTemp.SPStepLength, in2 := #SS_ParamTemp.SPStepLength)
   END_RUNG wire#w1
   RUNG wire#powerrail
      { S7_Templates := "SrcType := Int" } NE_Contact(in1 := #TS_ParamTemp.SPBurnerHigh, in2 := #SS_ParamTemp.SPBurnerHigh)
   END_RUNG wire#w1
   RUNG wire#powerrail
      { S7_Templates := "SrcType := Int" } NE_Contact(in1 := #TS_ParamTemp.SPTempSetpointZ1, in2 := #SS_ParamTemp.SPTempSetpointZ1)
   END_RUNG wire#w1
   RUNG wire#powerrail
      { S7_Templates := "SrcType := Int" } NE_Contact(in1 := #TS_ParamTemp.SPTempSetpointZ2, in2 := #SS_ParamTemp.SPTempSetpointZ2)
   END_RUNG wire#w1
   RUNG wire#powerrail
      { S7_Templates := "SrcType := Int" } NE_Contact(in1 := #TS_ParamTemp.SPTempSetpointZ3, in2 := #SS_ParamTemp.SPTempSetpointZ3)
   END_RUNG wire#w1
   RUNG wire#powerrail
      { S7_Templates := "SrcType := Int" } NE_Contact(in1 := #TS_ParamTemp.SPTempSetpointZ4, in2 := #SS_ParamTemp.SPTempSetpointZ4)
   END_RUNG wire#w1
   RUNG wire#powerrail
      { S7_Templates := "SrcType := Int" } NE_Contact(in1 := #TS_ParamTemp.SPTempSetpointZ5, in2 := #SS_ParamTemp.SPTempSetpointZ5)
   END_RUNG wire#w1
   // the same network as SCL:
   IF (#TS_ParamTemp.PartType <> #SS_ParamTemp.PartType) OR (#TS_ParamTemp.SPTactTime <> #SS_ParamTemp.SPTactTime) OR (#TS_ParamTemp.SPStepLength <> #SS_ParamTemp.SPStepLength) OR (#TS_ParamTemp.SPBurnerHigh <> #SS_ParamTemp.SPBurnerHigh) OR (#TS_ParamTemp.SPTempSetpointZ1 <> #SS_ParamTemp.SPTempSetpointZ1) OR (#TS_ParamTemp.SPTempSetpointZ2 <> #SS_ParamTemp.SPTempSetpointZ2) OR (#TS_ParamTemp.SPTempSetpointZ3 <> #SS_ParamTemp.SPTempSetpointZ3) OR (#TS_ParamTemp.SPTempSetpointZ4 <> #SS_ParamTemp.SPTempSetpointZ4) OR (#TS_ParamTemp.SPTempSetpointZ5 <> #SS_ParamTemp.SPTempSetpointZ5) THEN
       #SB1ParamChanged := TRUE;
   END_IF;
END_REGION

REGION Network 31: Production parameters values memory for next cycle evaluation
   RUNG wire#powerrail
      Move(in := #TS_ParamTemp.PartType, out1 => #SS_ParamTemp.PartType)
      Move(in := #TS_ParamTemp.SPTactTime, out1 => #SS_ParamTemp.SPTactTime)
      Move(in := #TS_ParamTemp.SPStepLength, out1 => #SS_ParamTemp.SPStepLength)
      Move(in := #TS_ParamTemp.SPBurnerHigh, out1 => #SS_ParamTemp.SPBurnerHigh)
   END_RUNG
   RUNG wire#powerrail
      Move(in := #TS_ParamTemp.SPTempSetpointZ1, out1 => #SS_ParamTemp.SPTempSetpointZ1)
      Move(in := #TS_ParamTemp.SPTempSetpointZ2, out1 => #SS_ParamTemp.SPTempSetpointZ2)
      Move(in := #TS_ParamTemp.SPTempSetpointZ3, out1 => #SS_ParamTemp.SPTempSetpointZ3)
   END_RUNG
   RUNG wire#powerrail
      Move(in := #TS_ParamTemp.SPTempSetpointZ4, out1 => #SS_ParamTemp.SPTempSetpointZ4)
      Move(in := #TS_ParamTemp.SPTempSetpointZ5, out1 => #SS_ParamTemp.SPTempSetpointZ5)
   END_RUNG
   // the same network as SCL:
   #SS_ParamTemp.PartType := #TS_ParamTemp.PartType;
   #SS_ParamTemp.SPTactTime := #TS_ParamTemp.SPTactTime;
   #SS_ParamTemp.SPStepLength := #TS_ParamTemp.SPStepLength;
   #SS_ParamTemp.SPBurnerHigh := #TS_ParamTemp.SPBurnerHigh;
   #SS_ParamTemp.SPTempSetpointZ1 := #TS_ParamTemp.SPTempSetpointZ1;
   #SS_ParamTemp.SPTempSetpointZ2 := #TS_ParamTemp.SPTempSetpointZ2;
   #SS_ParamTemp.SPTempSetpointZ3 := #TS_ParamTemp.SPTempSetpointZ3;
   #SS_ParamTemp.SPTempSetpointZ4 := #TS_ParamTemp.SPTempSetpointZ4;
   #SS_ParamTemp.SPTempSetpointZ5 := #TS_ParamTemp.SPTempSetpointZ5;
END_REGION

REGION Network 32: Send production parameters to owens PLC
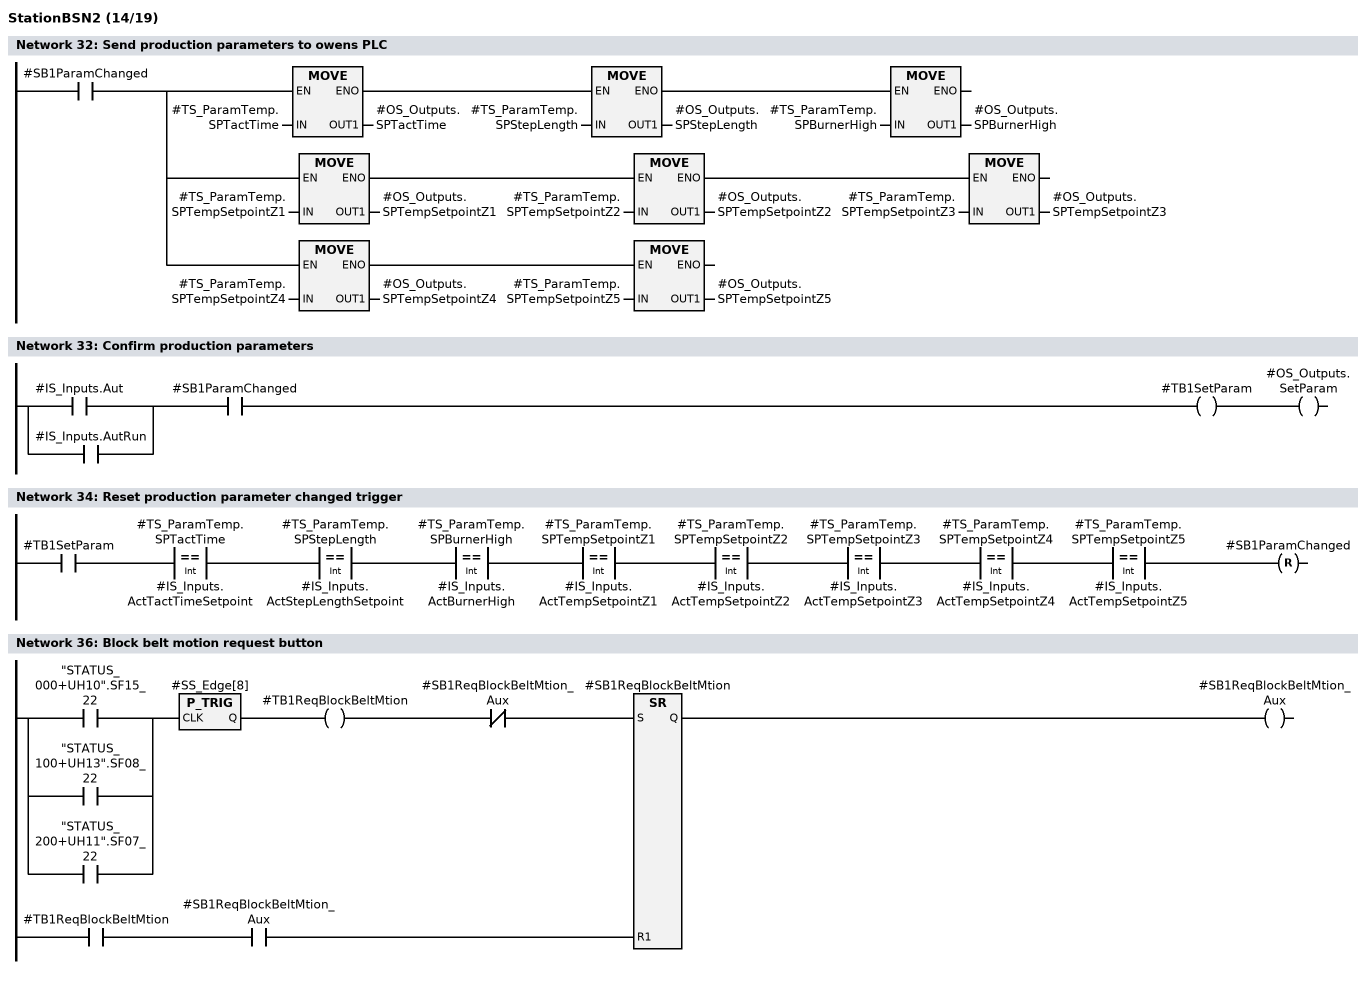
   RUNG wire#powerrail
      Contact( #SB1ParamChanged )
      wire#w1
      Move(in := #TS_ParamTemp.SPTactTime, out1 => #OS_Outputs.SPTactTime)
      Move(in := #TS_ParamTemp.SPStepLength, out1 => #OS_Outputs.SPStepLength)
      Move(in := #TS_ParamTemp.SPBurnerHigh, out1 => #OS_Outputs.SPBurnerHigh)
   END_RUNG
   RUNG wire#w1
      Move(in := #TS_ParamTemp.SPTempSetpointZ1, out1 => #OS_Outputs.SPTempSetpointZ1)
      Move(in := #TS_ParamTemp.SPTempSetpointZ2, out1 => #OS_Outputs.SPTempSetpointZ2)
      Move(in := #TS_ParamTemp.SPTempSetpointZ3, out1 => #OS_Outputs.SPTempSetpointZ3)
   END_RUNG
   RUNG wire#w1
      Move(in := #TS_ParamTemp.SPTempSetpointZ4, out1 => #OS_Outputs.SPTempSetpointZ4)
      Move(in := #TS_ParamTemp.SPTempSetpointZ5, out1 => #OS_Outputs.SPTempSetpointZ5)
   END_RUNG
   // the same network as SCL:
   IF #SB1ParamChanged THEN
       #OS_Outputs.SPTactTime := #TS_ParamTemp.SPTactTime;
       #OS_Outputs.SPStepLength := #TS_ParamTemp.SPStepLength;
       #OS_Outputs.SPBurnerHigh := #TS_ParamTemp.SPBurnerHigh;
       #OS_Outputs.SPTempSetpointZ1 := #TS_ParamTemp.SPTempSetpointZ1;
       #OS_Outputs.SPTempSetpointZ2 := #TS_ParamTemp.SPTempSetpointZ2;
       #OS_Outputs.SPTempSetpointZ3 := #TS_ParamTemp.SPTempSetpointZ3;
       #OS_Outputs.SPTempSetpointZ4 := #TS_ParamTemp.SPTempSetpointZ4;
       #OS_Outputs.SPTempSetpointZ5 := #TS_ParamTemp.SPTempSetpointZ5;
   END_IF;
END_REGION

REGION Network 33: Confirm production parameters
   RUNG wire#powerrail
      Contact( #IS_Inputs.Aut )
      wire#w1
      Contact( #SB1ParamChanged )
      Coil( #TB1SetParam )
      Coil( #OS_Outputs.SetParam )
   END_RUNG
   RUNG wire#powerrail
      Contact( #IS_Inputs.AutRun )
   END_RUNG wire#w1
   // the same network as SCL:
   #TB1SetParam := (#IS_Inputs.Aut OR #IS_Inputs.AutRun) AND #SB1ParamChanged;
   #OS_Outputs.SetParam := #TB1SetParam;
END_REGION

REGION Network 34: Reset production parameter changed trigger
   RUNG wire#powerrail
      Contact( #TB1SetParam )
      { S7_Templates := "SrcType := Int" } EQ_Contact(in1 := #TS_ParamTemp.SPTactTime, in2 := #IS_Inputs.ActTactTimeSetpoint)
      { S7_Templates := "SrcType := Int" } EQ_Contact(in1 := #TS_ParamTemp.SPStepLength, in2 := #IS_Inputs.ActStepLengthSetpoint)
      { S7_Templates := "SrcType := Int" } EQ_Contact(in1 := #TS_ParamTemp.SPBurnerHigh, in2 := #IS_Inputs.ActBurnerHigh)
      { S7_Templates := "SrcType := Int" } EQ_Contact(in1 := #TS_ParamTemp.SPTempSetpointZ1, in2 := #IS_Inputs.ActTempSetpointZ1)
      { S7_Templates := "SrcType := Int" } EQ_Contact(in1 := #TS_ParamTemp.SPTempSetpointZ2, in2 := #IS_Inputs.ActTempSetpointZ2)
      { S7_Templates := "SrcType := Int" } EQ_Contact(in1 := #TS_ParamTemp.SPTempSetpointZ3, in2 := #IS_Inputs.ActTempSetpointZ3)
      { S7_Templates := "SrcType := Int" } EQ_Contact(in1 := #TS_ParamTemp.SPTempSetpointZ4, in2 := #IS_Inputs.ActTempSetpointZ4)
      { S7_Templates := "SrcType := Int" } EQ_Contact(in1 := #TS_ParamTemp.SPTempSetpointZ5, in2 := #IS_Inputs.ActTempSetpointZ5)
      R_Coil( #SB1ParamChanged )
   END_RUNG
   // the same network as SCL:
   IF #TB1SetParam AND (#TS_ParamTemp.SPTactTime = #IS_Inputs.ActTactTimeSetpoint) AND (#TS_ParamTemp.SPStepLength = #IS_Inputs.ActStepLengthSetpoint) AND (#TS_ParamTemp.SPBurnerHigh = #IS_Inputs.ActBurnerHigh) AND (#TS_ParamTemp.SPTempSetpointZ1 = #IS_Inputs.ActTempSetpointZ1) AND (#TS_ParamTemp.SPTempSetpointZ2 = #IS_Inputs.ActTempSetpointZ2) AND (#TS_ParamTemp.SPTempSetpointZ3 = #IS_Inputs.ActTempSetpointZ3) AND (#TS_ParamTemp.SPTempSetpointZ4 = #IS_Inputs.ActTempSetpointZ4) AND (#TS_ParamTemp.SPTempSetpointZ5 = #IS_Inputs.ActTempSetpointZ5) THEN
       #SB1ParamChanged := FALSE;
   END_IF;
END_REGION

REGION Network 35: *************** Belt ***************
END_REGION

REGION Network 36: Block belt motion request button
   RUNG wire#powerrail
      Contact( "STATUS_000+UH10".SF15_22 )
      wire#w1
      P_Trig( #SS_Edge[8] )
      Coil( #TB1ReqBlockBeltMtion )
      I_Contact( #SB1ReqBlockBeltMtion_Aux )
      S_SR(operand := #SB1ReqBlockBeltMtion, r1 := wire#w2)
      Coil( #SB1ReqBlockBeltMtion_Aux )
   END_RUNG
   RUNG wire#powerrail
      Contact( "STATUS_100+UH13".SF08_22 )
   END_RUNG wire#w1
   RUNG wire#powerrail
      Contact( "STATUS_200+UH11".SF07_22 )
   END_RUNG wire#w1
   RUNG wire#powerrail
      Contact( #TB1ReqBlockBeltMtion )
      Contact( #SB1ReqBlockBeltMtion_Aux )
   END_RUNG wire#w2
   // the same network as SCL:
   #_w1 := "STATUS_000+UH10".SF15_22 OR "STATUS_100+UH13".SF08_22 OR "STATUS_200+UH11".SF07_22;
   #_w2 := #_w1 AND NOT #SS_Edge[8];   // rising edge
   #SS_Edge[8] := #_w1;
   #TB1ReqBlockBeltMtion := #_w2;
   IF #_w2 AND NOT #SB1ReqBlockBeltMtion_Aux THEN
       #SB1ReqBlockBeltMtion := TRUE;   // SR flip-flop
   END_IF;
   IF #TB1ReqBlockBeltMtion AND #SB1ReqBlockBeltMtion_Aux THEN #SB1ReqBlockBeltMtion := FALSE; END_IF;
   #SB1ReqBlockBeltMtion_Aux := #SB1ReqBlockBeltMtion;
END_REGION

REGION Network 37: Enable for robot 1R6 to enter zone BSN1
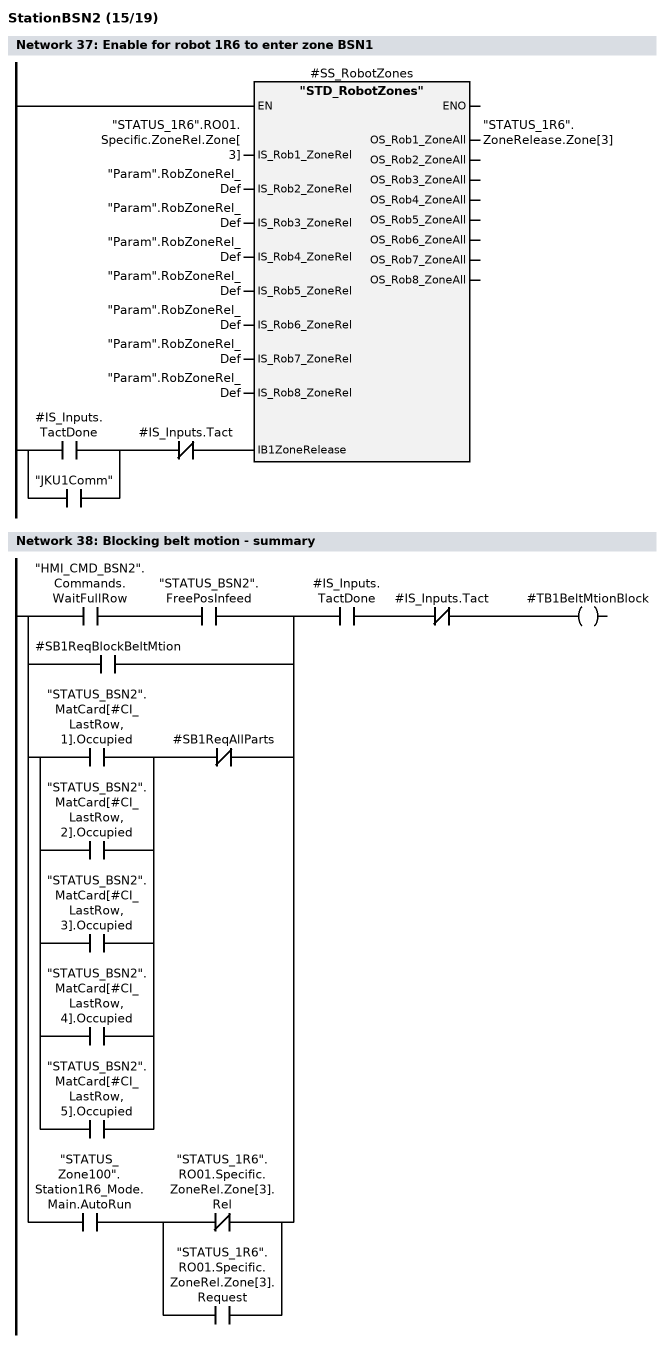
   RUNG wire#powerrail
      #SS_RobotZones(IB1ZoneRelease := wire#w2, IS_Rob1_ZoneRel := "STATUS_1R6".RO01.Specific.ZoneRel.Zone[3], IS_Rob2_ZoneRel := "Param".RobZoneRel_Def, IS_Rob3_ZoneRel := "Param".RobZoneRel_Def, IS_Rob4_ZoneRel := "Param".RobZoneRel_Def, IS_Rob5_ZoneRel := "Param".RobZoneRel_Def, IS_Rob6_ZoneRel := "Param".RobZoneRel_Def, IS_Rob7_ZoneRel := "Param".RobZoneRel_Def, IS_Rob8_ZoneRel := "Param".RobZoneRel_Def, OS_Rob1_ZoneAll => "STATUS_1R6".ZoneRelease.Zone[3], OS_Rob2_ZoneAll =>, OS_Rob3_ZoneAll =>, OS_Rob4_ZoneAll =>, OS_Rob5_ZoneAll =>, OS_Rob6_ZoneAll =>, OS_Rob7_ZoneAll =>, OS_Rob8_ZoneAll =>)
   END_RUNG
   RUNG wire#powerrail
      Contact( #IS_Inputs.TactDone )
      wire#w1
      I_Contact( #IS_Inputs.Tact )
   END_RUNG wire#w2
   RUNG wire#powerrail
      Contact( "JKU1Comm" )
   END_RUNG wire#w1
   // the same network as SCL:
   #SS_RobotZones(IS_Rob1_ZoneRel := "STATUS_1R6".RO01.Specific.ZoneRel.Zone[3],   // "STD_RobotZones"
                  IS_Rob2_ZoneRel := "Param".RobZoneRel_Def,
                  IS_Rob3_ZoneRel := "Param".RobZoneRel_Def,
                  IS_Rob4_ZoneRel := "Param".RobZoneRel_Def,
                  IS_Rob5_ZoneRel := "Param".RobZoneRel_Def,
                  IS_Rob6_ZoneRel := "Param".RobZoneRel_Def,
                  IS_Rob7_ZoneRel := "Param".RobZoneRel_Def,
                  IS_Rob8_ZoneRel := "Param".RobZoneRel_Def,
                  IB1ZoneRelease := (#IS_Inputs.TactDone OR "JKU1Comm") AND NOT #IS_Inputs.Tact,
                  OS_Rob1_ZoneAll => "STATUS_1R6".ZoneRelease.Zone[3]);
END_REGION

REGION Network 38: Blocking belt motion - summary
   RUNG wire#powerrail
      Contact( "HMI_CMD_BSN2".Commands.WaitFullRow )
      Contact( "STATUS_BSN2".FreePosInfeed )
      wire#w1
      Contact( #IS_Inputs.TactDone )
      I_Contact( #IS_Inputs.Tact )
      Coil( #TB1BeltMtionBlock )
   END_RUNG
   RUNG wire#powerrail
      Contact( #SB1ReqBlockBeltMtion )
   END_RUNG wire#w1
   RUNG wire#powerrail
      Contact( "STATUS_BSN2".MatCard[#CI_LastRow, 1].Occupied )
      wire#w2
      I_Contact( #SB1ReqAllParts )
   END_RUNG wire#w1
   RUNG wire#powerrail
      Contact( "STATUS_BSN2".MatCard[#CI_LastRow, 2].Occupied )
   END_RUNG wire#w2
   RUNG wire#powerrail
      Contact( "STATUS_BSN2".MatCard[#CI_LastRow, 3].Occupied )
   END_RUNG wire#w2
   RUNG wire#powerrail
      Contact( "STATUS_BSN2".MatCard[#CI_LastRow, 4].Occupied )
   END_RUNG wire#w2
   RUNG wire#powerrail
      Contact( "STATUS_BSN2".MatCard[#CI_LastRow, 5].Occupied )
   END_RUNG wire#w2
   RUNG wire#powerrail
      Contact( "STATUS_Zone100".Station1R6_Mode.Main.AutoRun )
      wire#w3
      I_Contact( "STATUS_1R6".RO01.Specific.ZoneRel.Zone[3].Rel )
   END_RUNG wire#w1
   RUNG wire#w3
      Contact( "STATUS_1R6".RO01.Specific.ZoneRel.Zone[3].Request )
   END_RUNG wire#w1
   // the same network as SCL:
   #TB1BeltMtionBlock := (("HMI_CMD_BSN2".Commands.WaitFullRow AND "STATUS_BSN2".FreePosInfeed) OR #SB1ReqBlockBeltMtion OR (("STATUS_BSN2".MatCard[#CI_LastRow, 1].Occupied OR "STATUS_BSN2".MatCard[#CI_LastRow, 2].Occupied OR "STATUS_BSN2".MatCard[#CI_LastRow, 3].Occupied OR "STATUS_BSN2".MatCard[#CI_LastRow, 4].Occupied OR "STATUS_BSN2".MatCard[#CI_LastRow, 5].Occupied) AND NOT #SB1ReqAllParts) OR ("STATUS_Zone100".Station1R6_Mode.Main.AutoRun AND (NOT "STATUS_1R6".RO01.Specific.ZoneRel.Zone[3].Rel OR "STATUS_1R6".RO01.Specific.ZoneRel.Zone[3].Request))) AND #IS_Inputs.TactDone AND NOT #IS_Inputs.Tact;
END_REGION

REGION Network 39: Belt motion enable
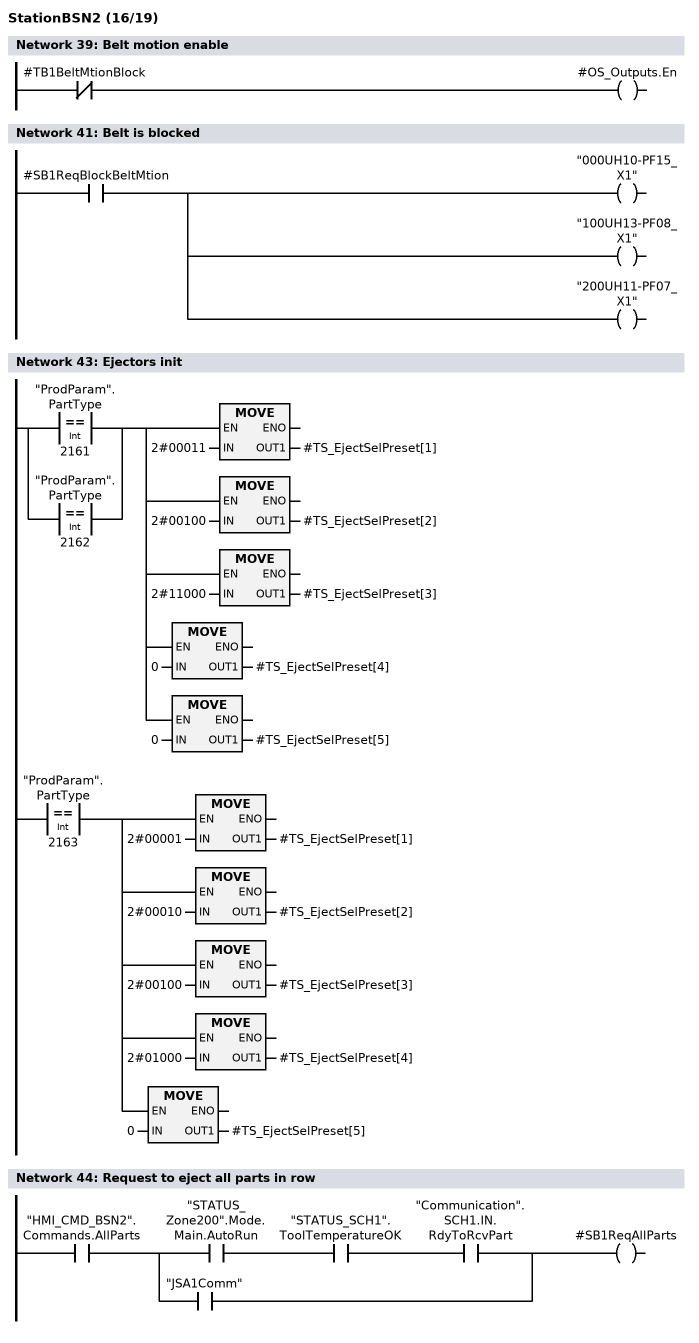
   RUNG wire#powerrail
      I_Contact( #TB1BeltMtionBlock )
      Coil( #OS_Outputs.En )
   END_RUNG
   // the same network as SCL:
   #OS_Outputs.En := NOT #TB1BeltMtionBlock;
END_REGION

REGION Network 40: ************** Signalization ***************
END_REGION

REGION Network 41: Belt is blocked
   RUNG wire#powerrail
      Contact( #SB1ReqBlockBeltMtion )
      wire#w1
      Coil( "000UH10-PF15_X1" )
   END_RUNG
   RUNG wire#w1
      Coil( "100UH13-PF08_X1" )
   END_RUNG
   RUNG wire#w1
      Coil( "200UH11-PF07_X1" )
   END_RUNG
   // the same network as SCL:
   "000UH10-PF15_X1" := #SB1ReqBlockBeltMtion;
   "100UH13-PF08_X1" := #SB1ReqBlockBeltMtion;
   "200UH11-PF07_X1" := #SB1ReqBlockBeltMtion;
END_REGION

REGION Network 42: *************** Ejectors ***************
END_REGION

REGION Network 43: Ejectors init
   RUNG wire#powerrail
      { S7_Templates := "SrcType := Int" } EQ_Contact(in1 := "ProdParam".PartType, in2 := 2161)
      wire#w1
      Move(in := 2#00011, out1 => #TS_EjectSelPreset[1])
   END_RUNG
   RUNG wire#powerrail
      { S7_Templates := "SrcType := Int" } EQ_Contact(in1 := "ProdParam".PartType, in2 := 2162)
   END_RUNG wire#w1
   RUNG wire#w1
      Move(in := 2#00100, out1 => #TS_EjectSelPreset[2])
   END_RUNG
   RUNG wire#w1
      Move(in := 2#11000, out1 => #TS_EjectSelPreset[3])
   END_RUNG
   RUNG wire#w1
      Move(in := 0, out1 => #TS_EjectSelPreset[4])
   END_RUNG
   RUNG wire#w1
      Move(in := 0, out1 => #TS_EjectSelPreset[5])
   END_RUNG
   RUNG wire#powerrail
      { S7_Templates := "SrcType := Int" } EQ_Contact(in1 := "ProdParam".PartType, in2 := 2163)
      wire#w2
      Move(in := 2#00001, out1 => #TS_EjectSelPreset[1])
   END_RUNG
   RUNG wire#w2
      Move(in := 2#00010, out1 => #TS_EjectSelPreset[2])
   END_RUNG
   RUNG wire#w2
      Move(in := 2#00100, out1 => #TS_EjectSelPreset[3])
   END_RUNG
   RUNG wire#w2
      Move(in := 2#01000, out1 => #TS_EjectSelPreset[4])
   END_RUNG
   RUNG wire#w2
      Move(in := 0, out1 => #TS_EjectSelPreset[5])
   END_RUNG
   // the same network as SCL:
   IF ("ProdParam".PartType = 2161) OR ("ProdParam".PartType = 2162) THEN
       #TS_EjectSelPreset[1] := 2#00011;
       #TS_EjectSelPreset[2] := 2#00100;
       #TS_EjectSelPreset[3] := 2#11000;
       #TS_EjectSelPreset[4] := 0;
       #TS_EjectSelPreset[5] := 0;
   END_IF;
   IF "ProdParam".PartType = 2163 THEN
       #TS_EjectSelPreset[1] := 2#00001;
       #TS_EjectSelPreset[2] := 2#00010;
       #TS_EjectSelPreset[3] := 2#00100;
       #TS_EjectSelPreset[4] := 2#01000;
       #TS_EjectSelPreset[5] := 0;
   END_IF;
END_REGION

REGION Network 44: Request to eject all parts in row
   RUNG wire#powerrail
      Contact( "HMI_CMD_BSN2".Commands.AllParts )
      wire#w1
      Contact( "STATUS_Zone200".Mode.Main.AutoRun )
      Contact( "STATUS_SCH1".ToolTemperatureOK )
      Contact( "Communication".SCH1.IN.RdyToRcvPart )
      wire#w2
      Coil( #SB1ReqAllParts )
   END_RUNG
   RUNG wire#w1
      Contact( "JSA1Comm" )
   END_RUNG wire#w2
   // the same network as SCL:
   #SB1ReqAllParts := "HMI_CMD_BSN2".Commands.AllParts AND (("STATUS_Zone200".Mode.Main.AutoRun AND "STATUS_SCH1".ToolTemperatureOK AND "Communication".SCH1.IN.RdyToRcvPart) OR "JSA1Comm");
END_REGION

REGION Network 45: Open doors when request to eject all parts in row + part presented + belt step started
   // #SS_Edge[6] - open door request to owen
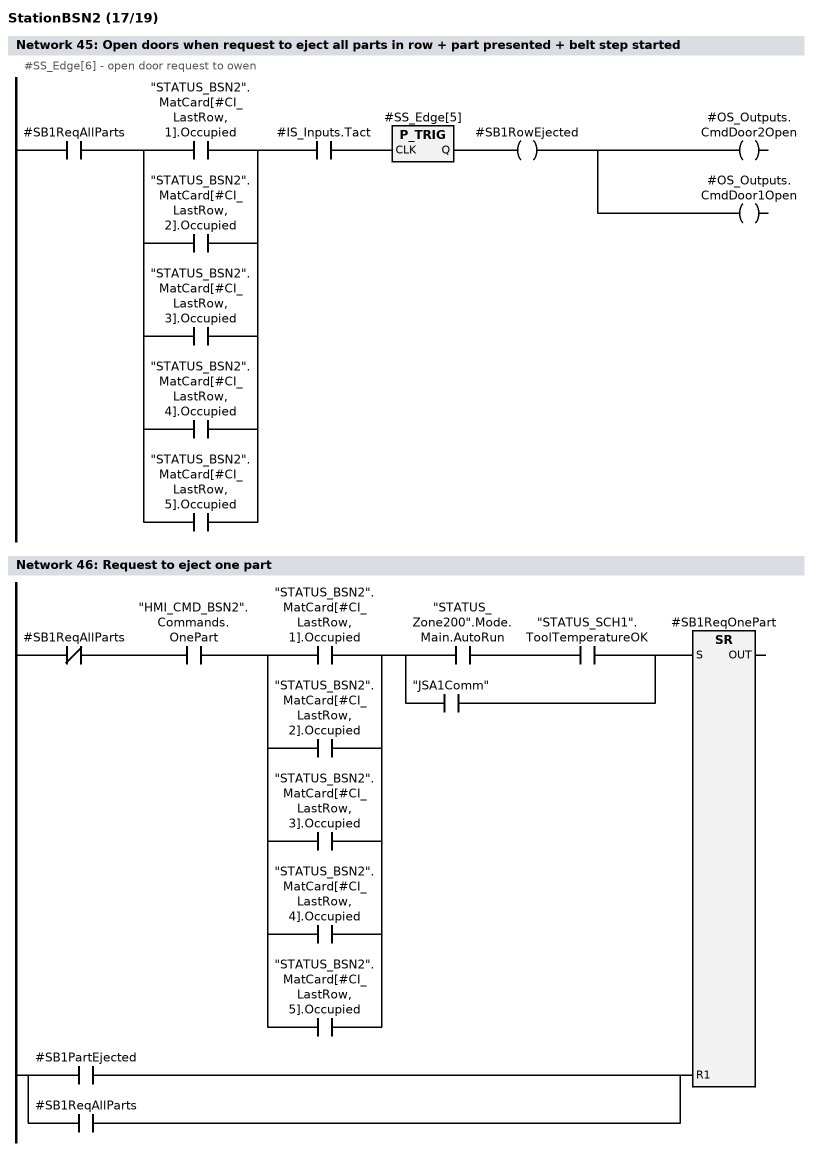
   RUNG wire#powerrail
      Contact( #SB1ReqAllParts )
      wire#w1
      Contact( "STATUS_BSN2".MatCard[#CI_LastRow, 1].Occupied )
      wire#w2
      Contact( #IS_Inputs.Tact )
      P_Trig( #SS_Edge[5] )
      Coil( #SB1RowEjected )
      wire#w3
      Coil( #OS_Outputs.CmdDoor2Open )
   END_RUNG
   RUNG wire#w1
      Contact( "STATUS_BSN2".MatCard[#CI_LastRow, 2].Occupied )
   END_RUNG wire#w2
   RUNG wire#w1
      Contact( "STATUS_BSN2".MatCard[#CI_LastRow, 3].Occupied )
   END_RUNG wire#w2
   RUNG wire#w1
      Contact( "STATUS_BSN2".MatCard[#CI_LastRow, 4].Occupied )
   END_RUNG wire#w2
   RUNG wire#w1
      Contact( "STATUS_BSN2".MatCard[#CI_LastRow, 5].Occupied )
   END_RUNG wire#w2
   RUNG wire#w3
      Coil( #OS_Outputs.CmdDoor1Open )
   END_RUNG
   // the same network as SCL:
   #_w1 := #SB1ReqAllParts AND ("STATUS_BSN2".MatCard[#CI_LastRow, 1].Occupied OR "STATUS_BSN2".MatCard[#CI_LastRow, 2].Occupied OR "STATUS_BSN2".MatCard[#CI_LastRow, 3].Occupied OR "STATUS_BSN2".MatCard[#CI_LastRow, 4].Occupied OR "STATUS_BSN2".MatCard[#CI_LastRow, 5].Occupied) AND #IS_Inputs.Tact;
   #_w2 := #_w1 AND NOT #SS_Edge[5];   // rising edge
   #SS_Edge[5] := #_w1;
   #SB1RowEjected := #_w2;
   #OS_Outputs.CmdDoor2Open := #_w2;
   #OS_Outputs.CmdDoor1Open := #_w2;
END_REGION

REGION Network 46: Request to eject one part
   RUNG wire#powerrail
      I_Contact( #SB1ReqAllParts )
      Contact( "HMI_CMD_BSN2".Commands.OnePart )
      wire#w1
      Contact( "STATUS_BSN2".MatCard[#CI_LastRow, 1].Occupied )
      wire#w2
      Contact( "STATUS_Zone200".Mode.Main.AutoRun )
      Contact( "STATUS_SCH1".ToolTemperatureOK )
      wire#w3
      S_SR(operand := #SB1ReqOnePart, r1 := wire#w4)
   END_RUNG
   RUNG wire#w1
      Contact( "STATUS_BSN2".MatCard[#CI_LastRow, 2].Occupied )
   END_RUNG wire#w2
   RUNG wire#w1
      Contact( "STATUS_BSN2".MatCard[#CI_LastRow, 3].Occupied )
   END_RUNG wire#w2
   RUNG wire#w1
      Contact( "STATUS_BSN2".MatCard[#CI_LastRow, 4].Occupied )
   END_RUNG wire#w2
   RUNG wire#w1
      Contact( "STATUS_BSN2".MatCard[#CI_LastRow, 5].Occupied )
   END_RUNG wire#w2
   RUNG wire#w2
      Contact( "JSA1Comm" )
   END_RUNG wire#w3
   RUNG wire#powerrail
      Contact( #SB1PartEjected )
   END_RUNG wire#w4
   RUNG wire#powerrail
      Contact( #SB1ReqAllParts )
   END_RUNG wire#w4
   // the same network as SCL:
   IF NOT #SB1ReqAllParts AND "HMI_CMD_BSN2".Commands.OnePart AND ("STATUS_BSN2".MatCard[#CI_LastRow, 1].Occupied OR "STATUS_BSN2".MatCard[#CI_LastRow, 2].Occupied OR "STATUS_BSN2".MatCard[#CI_LastRow, 3].Occupied OR "STATUS_BSN2".MatCard[#CI_LastRow, 4].Occupied OR "STATUS_BSN2".MatCard[#CI_LastRow, 5].Occupied) AND (("STATUS_Zone200".Mode.Main.AutoRun AND "STATUS_SCH1".ToolTemperatureOK) OR "JSA1Comm") THEN
       #SB1ReqOnePart := TRUE;   // SR flip-flop
   END_IF;
   IF #SB1PartEjected OR #SB1ReqAllParts THEN #SB1ReqOnePart := FALSE; END_IF;
END_REGION

